	garr_betriebsmeldungen[st_config.i16_meld_startindex + 0] := FALSE;
	garr_betriebsmeldungen[st_config.i16_meld_startindex + 1] := FALSE;
	garr_betriebsmeldungen[st_config.i16_meld_startindex + 2] := FALSE;
	garr_betriebsmeldungen[st_config.i16_meld_startindex + 3] := FALSE;
	garr_betriebsmeldungen[st_config.i16_meld_startindex + 4] := FALSE;
	garr_betriebsmeldungen[st_config.i16_meld_startindex + 5] := FALSE;
	garr_betriebsmeldungen[st_config.i16_meld_startindex + 6] := FALSE;
	garr_betriebsmeldungen[st_config.i16_meld_startindex + 7] := FALSE;
	garr_betriebsmeldungen[st_config.i16_meld_startindex + 8] := FALSE;
	garr_betriebsmeldungen[st_config.i16_meld_startindex + 9] := FALSE;
	garr_betriebsmeldungen[st_config.i16_meld_startindex + 10] := FALSE;
	garr_betriebsmeldungen[st_config.i16_meld_startindex + 11] := FALSE;
	garr_betriebsmeldungen[st_config.i16_meld_startindex + 12] := FALSE;
	garr_betriebsmeldungen[st_config.i16_meld_startindex + 13] := FALSE;
	garr_betriebsmeldungen[st_config.i16_meld_startindex + 14] := FALSE;
	garr_betriebsmeldungen[st_config.i16_meld_startindex + 15] := FALSE;
	garr_betriebsmeldungen[st_config.i16_meld_startindex + 16] := FALSE;
	garr_betriebsmeldungen[st_config.i16_meld_startindex + 17] := FALSE;
	garr_betriebsmeldungen[st_config.i16_meld_startindex + 18] := FALSE;
	garr_betriebsmeldungen[st_config.i16_meld_startindex + 19] := FALSE;
END_IF
END_PROGRAM

(* POU Gemeinsamkeiten17xx/Zylinder/ST_Zylinder, ST *)
PROGRAM ST_Zylinder
VAR
	b_first_cycle 			: BOOL := TRUE;
END_VAR
IF ST_BBGen.b_lesen_komplett THEN

	ST_Datainit_Zylinder();

	(* Zylinderaufrufe *)
	zyl_wt_zentrierer_tisch.fb(
		st_config:= ,
		bw_nocken_zylinder_einfahren:= ,
		bw_nocken_zylinder_ausfahren:= ,
		uw_nocken_zylinder_einfahren:= ,
		uw_nocken_zylinder_ausfahren:= ,
		b_direkttaste_ausfahren:= ,
		b_direkttaste_mittefahren:= ,
		b_direkttaste_einfahren	:= ,
		e_druckwaechter:= ST_Betriebsfreigaben.e_druckwaechter,
		i16_betriebsart:= gi16_betriebsart,
		b_no_gesteuert_im_norm_betrieb:= ,
		st_ctrl_in:= zyl_wt_zentrierer_tisch.st_ctrl.in,
		b_masterachse_hand_dialog_aktiv:= ,
		st_visu:= visu.st_zyl,
		st_ctrl_out=> zyl_wt_zentrierer_tisch.st_ctrl.out,
		a_ventil_einfahren=> ,
		a_ventil_ausfahren=> );
	
	zyl_wt_stopper_tisch.fb(
		st_config:= ,
		bw_nocken_zylinder_einfahren:= ,
		bw_nocken_zylinder_ausfahren:= ,
		uw_nocken_zylinder_einfahren:= ,
		uw_nocken_zylinder_ausfahren:= ,
		b_direkttaste_ausfahren:= ,
		b_direkttaste_mittefahren:= ,
		b_direkttaste_einfahren	:= ,
		e_druckwaechter:= ST_Betriebsfreigaben.e_druckwaechter,
		i16_betriebsart:= gi16_betriebsart,
		b_no_gesteuert_im_norm_betrieb:= ,
		st_ctrl_in:= zyl_wt_stopper_tisch.st_ctrl.in,
		b_masterachse_hand_dialog_aktiv:= ,
		st_visu:= visu.st_zyl,
		st_ctrl_out=> zyl_wt_stopper_tisch.st_ctrl.out,
		a_ventil_einfahren=> ,
		a_ventil_ausfahren=> );
	
	zyl_wt_stopper_auslauf.fb(
		st_config:= ,
		bw_nocken_zylinder_einfahren:= ,
		bw_nocken_zylinder_ausfahren:= ,
		uw_nocken_zylinder_einfahren:= ,
		uw_nocken_zylinder_ausfahren:= ,
		b_direkttaste_ausfahren:= ,
		b_direkttaste_mittefahren:= ,
		b_direkttaste_einfahren	:= ,
		e_druckwaechter:= ST_Betriebsfreigaben.e_druckwaechter,
		i16_betriebsart:= gi16_betriebsart,
		b_no_gesteuert_im_norm_betrieb:= ,
		st_ctrl_in:= zyl_wt_stopper_auslauf.st_ctrl.in,
		b_masterachse_hand_dialog_aktiv:= ,
		st_visu:= visu.st_zyl,
		st_ctrl_out=> zyl_wt_stopper_auslauf.st_ctrl.out,
		a_ventil_einfahren=> ,
		a_ventil_ausfahren=> );
	
	zyl_hublift_rechts_lift.fb(
		st_config:= ,
		bw_nocken_zylinder_einfahren:= ,
		bw_nocken_zylinder_ausfahren:= ,
		uw_nocken_zylinder_einfahren:= ,
		uw_nocken_zylinder_ausfahren:= ,
		b_direkttaste_ausfahren:= ,
		b_direkttaste_mittefahren:= ,
		b_direkttaste_einfahren	:= ,
		e_druckwaechter:= ST_Betriebsfreigaben.e_druckwaechter,
		i16_betriebsart:= gi16_betriebsart,
		b_no_gesteuert_im_norm_betrieb:= ,
		st_ctrl_in:= zyl_hublift_rechts_lift.st_ctrl.in,
		b_masterachse_hand_dialog_aktiv:= ,
		st_visu:= visu.st_zyl,
		st_ctrl_out=> zyl_hublift_rechts_lift.st_ctrl.out,
		a_ventil_einfahren=> ,
		a_ventil_ausfahren=> );
	
	zyl_hublift_rechts_wt_einzug.fb(
		st_config:= ,
		bw_nocken_zylinder_einfahren:= ,
		bw_nocken_zylinder_ausfahren:= ,
		uw_nocken_zylinder_einfahren:= ,
		uw_nocken_zylinder_ausfahren:= ,
		b_direkttaste_ausfahren:= ,
		b_direkttaste_mittefahren:= ,
		b_direkttaste_einfahren	:= ,
		e_druckwaechter:= ST_Betriebsfreigaben.e_druckwaechter,
		i16_betriebsart:= gi16_betriebsart,
		b_no_gesteuert_im_norm_betrieb:= ,
		st_ctrl_in:= zyl_hublift_rechts_wt_einzug.st_ctrl.in,
		b_masterachse_hand_dialog_aktiv:= ,
		st_visu:= visu.st_zyl,
		st_ctrl_out=> zyl_hublift_rechts_wt_einzug.st_ctrl.out,
		a_ventil_einfahren=> ,
		a_ventil_ausfahren=> );
	
	zyl_hublift_rechts_wt_klinke.fb(
		st_config:= ,
		bw_nocken_zylinder_einfahren:= ,
		bw_nocken_zylinder_ausfahren:= ,
		uw_nocken_zylinder_einfahren:= ,
		uw_nocken_zylinder_ausfahren:= ,
		b_direkttaste_ausfahren:= ,
		b_direkttaste_mittefahren:= ,
		b_direkttaste_einfahren	:= ,
		e_druckwaechter:= ST_Betriebsfreigaben.e_druckwaechter,
		i16_betriebsart:= gi16_betriebsart,
		b_no_gesteuert_im_norm_betrieb:= ,
		st_ctrl_in:= zyl_hublift_rechts_wt_klinke.st_ctrl.in,
		b_masterachse_hand_dialog_aktiv:= ,
		st_visu:= visu.st_zyl,
		st_ctrl_out=> zyl_hublift_rechts_wt_klinke.st_ctrl.out,
		a_ventil_einfahren=> ,
		a_ventil_ausfahren=> );
	
	zyl_hublift_links_lift.fb(
		st_config:= ,
		bw_nocken_zylinder_einfahren:= ,
		bw_nocken_zylinder_ausfahren:= ,
		uw_nocken_zylinder_einfahren:= ,
		uw_nocken_zylinder_ausfahren:= ,
		b_direkttaste_ausfahren:= ,
		b_direkttaste_mittefahren:= ,
		b_direkttaste_einfahren	:= ,
		e_druckwaechter:= ST_Betriebsfreigaben.e_druckwaechter,
		i16_betriebsart:= gi16_betriebsart,
		b_no_gesteuert_im_norm_betrieb:= ,
		st_ctrl_in:= zyl_hublift_links_lift.st_ctrl.in,
		b_masterachse_hand_dialog_aktiv:= ,
		st_visu:= visu.st_zyl,
		st_ctrl_out=> zyl_hublift_links_lift.st_ctrl.out,
		a_ventil_einfahren=> ,
		a_ventil_ausfahren=> );
	
	zyl_hublift_links_wt_einzug.fb(
		st_config:= ,
		bw_nocken_zylinder_einfahren:= ,
		bw_nocken_zylinder_ausfahren:= ,
		uw_nocken_zylinder_einfahren:= ,
		uw_nocken_zylinder_ausfahren:= ,
		b_direkttaste_ausfahren:= ,
		b_direkttaste_mittefahren:= ,
		b_direkttaste_einfahren	:= ,
		e_druckwaechter:= ST_Betriebsfreigaben.e_druckwaechter,
		i16_betriebsart:= gi16_betriebsart,
		b_no_gesteuert_im_norm_betrieb:= ,
		st_ctrl_in:= zyl_hublift_links_wt_einzug.st_ctrl.in,
		b_masterachse_hand_dialog_aktiv:= ,
		st_visu:= visu.st_zyl,
		st_ctrl_out=> zyl_hublift_links_wt_einzug.st_ctrl.out,
		a_ventil_einfahren=> ,
		a_ventil_ausfahren=> );
	
	zyl_hublift_links_wt_klinke.fb(
		st_config:= ,
		bw_nocken_zylinder_einfahren:= ,
		bw_nocken_zylinder_ausfahren:= ,
		uw_nocken_zylinder_einfahren:= ,
		uw_nocken_zylinder_ausfahren:= ,
		b_direkttaste_ausfahren:= ,
		b_direkttaste_mittefahren:= ,
		b_direkttaste_einfahren	:= ,
		e_druckwaechter:= ST_Betriebsfreigaben.e_druckwaechter,
		i16_betriebsart:= gi16_betriebsart,
		b_no_gesteuert_im_norm_betrieb:= ,
		st_ctrl_in:= zyl_hublift_links_wt_klinke.st_ctrl.in,
		b_masterachse_hand_dialog_aktiv:= ,
		st_visu:= visu.st_zyl,
		st_ctrl_out=> zyl_hublift_links_wt_klinke.st_ctrl.out,
		a_ventil_einfahren=> ,
		a_ventil_ausfahren=> );
	
	zyl_hublift_links_stopper.fb(
		st_config:= ,
		bw_nocken_zylinder_einfahren:= ,
		bw_nocken_zylinder_ausfahren:= ,
		uw_nocken_zylinder_einfahren:= ,
		uw_nocken_zylinder_ausfahren:= ,
		b_direkttaste_ausfahren:= ,
		b_direkttaste_mittefahren:= ,
		b_direkttaste_einfahren	:= ,
		e_druckwaechter:= ST_Betriebsfreigaben.e_druckwaechter,
		i16_betriebsart:= gi16_betriebsart,
		b_no_gesteuert_im_norm_betrieb:= ,
		st_ctrl_in:= zyl_hublift_links_stopper.st_ctrl.in,
		b_masterachse_hand_dialog_aktiv:= ,
		st_visu:= visu.st_zyl,
		st_ctrl_out=> zyl_hublift_links_stopper.st_ctrl.out,
		a_ventil_einfahren=> ,
		a_ventil_ausfahren=> );
	
	zyl_hublift_links_eingriffschutz.fb(
		st_config:= ,
		bw_nocken_zylinder_einfahren:= ,
		bw_nocken_zylinder_ausfahren:= ,
		uw_nocken_zylinder_einfahren:= ,
		uw_nocken_zylinder_ausfahren:= ,
		b_direkttaste_ausfahren:= ,
		b_direkttaste_mittefahren:= ,
		b_direkttaste_einfahren	:= ,
		e_druckwaechter:= ST_Betriebsfreigaben.e_druckwaechter,
		i16_betriebsart:= gi16_betriebsart,
		b_no_gesteuert_im_norm_betrieb:= ,
		st_ctrl_in:= zyl_hublift_links_eingriffschutz.st_ctrl.in,
		b_masterachse_hand_dialog_aktiv:= ,
		st_visu:= visu.st_zyl,
		st_ctrl_out=> zyl_hublift_links_eingriffschutz.st_ctrl.out,
		a_ventil_einfahren=> ,
		a_ventil_ausfahren=> );
	
	CASE gst_datensatz.st_md.i16_typ_zelle OF
		KEINE_ZELLE:
			;
	
		BESTUECKZELLE_1700:
			zyl_bawe_faenger_li.fb.st_config.b_aktiv := NOT gst_datensatz.st_md.b_wt_transport_simulation;
			zyl_bawe_faenger_li.fb(
				st_config:= ,
				bw_nocken_zylinder_einfahren:= ,
				bw_nocken_zylinder_ausfahren:= ,
				uw_nocken_zylinder_einfahren:= ,
				uw_nocken_zylinder_ausfahren:= ,
				b_direkttaste_ausfahren:= ,
				b_direkttaste_mittefahren:= ,
				b_direkttaste_einfahren	:= ,
				e_druckwaechter:= ST_Betriebsfreigaben.e_druckwaechter,
				i16_betriebsart:= gi16_betriebsart,
				b_no_gesteuert_im_norm_betrieb:= ,
				st_ctrl_in:= zyl_bawe_faenger_li.st_ctrl.in,
				b_masterachse_hand_dialog_aktiv:= ,
				st_visu:= visu.st_zyl,
				st_ctrl_out=> zyl_bawe_faenger_li.st_ctrl.out,
				a_ventil_einfahren=> ,
				a_ventil_ausfahren=> );
	
			zyl_bawe_faenger_re.fb.st_config.b_aktiv := NOT gst_datensatz.st_md.b_wt_transport_simulation;
			zyl_bawe_faenger_re.fb(
				st_config:= ,
				bw_nocken_zylinder_einfahren:= ,
				bw_nocken_zylinder_ausfahren:= ,
				uw_nocken_zylinder_einfahren:= ,
				uw_nocken_zylinder_ausfahren:= ,
				b_direkttaste_ausfahren:= ,
				b_direkttaste_mittefahren:= ,
				b_direkttaste_einfahren	:= ,
				e_druckwaechter:= ST_Betriebsfreigaben.e_druckwaechter,
				i16_betriebsart:= gi16_betriebsart,
				b_no_gesteuert_im_norm_betrieb:= ,
				st_ctrl_in:= zyl_bawe_faenger_re.st_ctrl.in,
				b_masterachse_hand_dialog_aktiv:= ,
				st_visu:= visu.st_zyl,
				st_ctrl_out=> zyl_bawe_faenger_re.st_ctrl.out,
				a_ventil_einfahren=> ,
				a_ventil_ausfahren=> );
	
			zyl_bawe_halter_li.fb.st_config.b_aktiv := NOT gst_datensatz.st_md.b_wt_transport_simulation;
			zyl_bawe_halter_li.fb(
				st_config:= ,
				bw_nocken_zylinder_einfahren:= ,
				bw_nocken_zylinder_ausfahren:= ,
				uw_nocken_zylinder_einfahren:= ,
				uw_nocken_zylinder_ausfahren:= ,
				b_direkttaste_ausfahren:= ,
				b_direkttaste_mittefahren:= ,
				b_direkttaste_einfahren	:= ,
				e_druckwaechter:= ST_Betriebsfreigaben.e_druckwaechter,
				i16_betriebsart:= gi16_betriebsart,
				b_no_gesteuert_im_norm_betrieb:= ,
				st_ctrl_in:= zyl_bawe_halter_li.st_ctrl.in,
				b_masterachse_hand_dialog_aktiv:= ,
				st_visu:= visu.st_zyl,
				st_ctrl_out=> zyl_bawe_halter_li.st_ctrl.out,
				a_ventil_einfahren=> ,
				a_ventil_ausfahren=> );
	
			zyl_bawe_halter_re.fb.st_config.b_aktiv := NOT gst_datensatz.st_md.b_wt_transport_simulation;
			zyl_bawe_halter_re.fb(
				st_config:= ,
				bw_nocken_zylinder_einfahren:= ,
				bw_nocken_zylinder_ausfahren:= ,
				uw_nocken_zylinder_einfahren:= ,
				uw_nocken_zylinder_ausfahren:= ,
				b_direkttaste_ausfahren:= ,
				b_direkttaste_mittefahren:= ,
				b_direkttaste_einfahren	:= ,
				e_druckwaechter:= ST_Betriebsfreigaben.e_druckwaechter,
				i16_betriebsart:= gi16_betriebsart,
				b_no_gesteuert_im_norm_betrieb:= ,
				st_ctrl_in:= zyl_bawe_halter_re.st_ctrl.in,
				b_masterachse_hand_dialog_aktiv:= ,
				st_visu:= visu.st_zyl,
				st_ctrl_out=> zyl_bawe_halter_re.st_ctrl.out,
				a_ventil_einfahren=> ,
				a_ventil_ausfahren=> );
	
			zyl_bawe_querschub.fb.st_config.b_aktiv := NOT gst_datensatz.st_md.b_wt_transport_simulation;
			zyl_bawe_querschub.fb(
				st_config:= ,
				bw_nocken_zylinder_einfahren:= ,
				bw_nocken_zylinder_ausfahren:= ,
				uw_nocken_zylinder_einfahren:= ,
				uw_nocken_zylinder_ausfahren:= ,
				b_direkttaste_ausfahren:= ,
				b_direkttaste_mittefahren:= ,
				b_direkttaste_einfahren	:= ,
				e_druckwaechter:= ST_Betriebsfreigaben.e_druckwaechter,
				i16_betriebsart:= gi16_betriebsart,
				b_no_gesteuert_im_norm_betrieb:= ,
				st_ctrl_in:= zyl_bawe_querschub.st_ctrl.in,
				b_masterachse_hand_dialog_aktiv:= ,
				st_visu:= visu.st_zyl,
				st_ctrl_out=> zyl_bawe_querschub.st_ctrl.out,
				a_ventil_einfahren=> ,
				a_ventil_ausfahren=> );
	
			zyl_bawe_vorschub.fb.st_config.b_aktiv := NOT gst_datensatz.st_md.b_wt_transport_simulation;
			zyl_bawe_vorschub.fb(
				st_config:= ,
				bw_nocken_zylinder_einfahren:= ,
				bw_nocken_zylinder_ausfahren:= ,
				uw_nocken_zylinder_einfahren:= ,
				uw_nocken_zylinder_ausfahren:= ,
				b_direkttaste_ausfahren:= ,
				b_direkttaste_mittefahren:= ,
				b_direkttaste_einfahren	:= ,
				e_druckwaechter:= ST_Betriebsfreigaben.e_druckwaechter,
				i16_betriebsart:= gi16_betriebsart,
				b_no_gesteuert_im_norm_betrieb:= ,
				st_ctrl_in:= zyl_bawe_vorschub.st_ctrl.in,
				b_masterachse_hand_dialog_aktiv:= ,
				st_visu:= visu.st_zyl,
				st_ctrl_out=> zyl_bawe_vorschub.st_ctrl.out,
				a_ventil_einfahren=> a_zyl_vorschub_einfahren,
				a_ventil_ausfahren=> a_zyl_vorschub_ausfahren);
			
			zyl_haspel_li_heben.fb(
				st_config:= ,
				bw_nocken_zylinder_einfahren:= ,
				bw_nocken_zylinder_ausfahren:= ,
				uw_nocken_zylinder_einfahren:= ,
				uw_nocken_zylinder_ausfahren:= ,
				b_direkttaste_ausfahren:= ,
				b_direkttaste_mittefahren:= ,
				b_direkttaste_einfahren	:= ,
				e_druckwaechter:= ST_Betriebsfreigaben.e_druckwaechter,
				i16_betriebsart:= gi16_betriebsart,
				b_no_gesteuert_im_norm_betrieb:= ,
				st_ctrl_in:= zyl_haspel_li_heben.st_ctrl.in,
				b_masterachse_hand_dialog_aktiv:= ,
				st_visu:= visu.st_zyl,
				st_ctrl_out=> zyl_haspel_li_heben.st_ctrl.out,
				a_ventil_einfahren=> ,
				a_ventil_ausfahren=> );
	
			zyl_haspel_li_abspulen.fb(
				st_config:= ,
				bw_nocken_zylinder_einfahren:= ,
				bw_nocken_zylinder_ausfahren:= ,
				uw_nocken_zylinder_einfahren:= ,
				uw_nocken_zylinder_ausfahren:= ,
				b_direkttaste_ausfahren:= ,
				b_direkttaste_mittefahren:= ,
				b_direkttaste_einfahren	:= ,
				e_druckwaechter:= ST_Betriebsfreigaben.e_druckwaechter,
				i16_betriebsart:= gi16_betriebsart,
				b_no_gesteuert_im_norm_betrieb:= ,
				st_ctrl_in:= zyl_haspel_li_abspulen.st_ctrl.in,
				b_masterachse_hand_dialog_aktiv:= ,
				st_visu:= visu.st_zyl,
				st_ctrl_out=> zyl_haspel_li_abspulen.st_ctrl.out,
				a_ventil_einfahren=> ,
				a_ventil_ausfahren=> );
			
			zyl_haspel_li_sperren.fb(
				st_config:= ,
				bw_nocken_zylinder_einfahren:= ,
				bw_nocken_zylinder_ausfahren:= ,
				uw_nocken_zylinder_einfahren:= ,
				uw_nocken_zylinder_ausfahren:= ,
				b_direkttaste_ausfahren:= ,
				b_direkttaste_mittefahren:= ,
				b_direkttaste_einfahren	:= ,
				e_druckwaechter:= ST_Betriebsfreigaben.e_druckwaechter,
				i16_betriebsart:= gi16_betriebsart,
				b_no_gesteuert_im_norm_betrieb:= ,
				st_ctrl_in:= zyl_haspel_li_sperren.st_ctrl.in,
				b_masterachse_hand_dialog_aktiv:= ,
				st_visu:= visu.st_zyl,
				st_ctrl_out=> zyl_haspel_li_sperren.st_ctrl.out,
				a_ventil_einfahren=> ,
				a_ventil_ausfahren=> );
			
			zyl_haspel_re_heben.fb(
				st_config:= ,
				bw_nocken_zylinder_einfahren:= ,
				bw_nocken_zylinder_ausfahren:= ,
				uw_nocken_zylinder_einfahren:= ,
				uw_nocken_zylinder_ausfahren:= ,
				b_direkttaste_ausfahren:= ,
				b_direkttaste_mittefahren:= ,
				b_direkttaste_einfahren	:= ,
				e_druckwaechter:= ST_Betriebsfreigaben.e_druckwaechter,
				i16_betriebsart:= gi16_betriebsart,
				b_no_gesteuert_im_norm_betrieb:= ,
				st_ctrl_in:= zyl_haspel_re_heben.st_ctrl.in,
				b_masterachse_hand_dialog_aktiv:= ,
				st_visu:= visu.st_zyl,
				st_ctrl_out=> zyl_haspel_re_heben.st_ctrl.out,
				a_ventil_einfahren=> ,
				a_ventil_ausfahren=> );
			
			zyl_haspel_re_abspulen.fb(
				st_config:= ,
				bw_nocken_zylinder_einfahren:= ,
				bw_nocken_zylinder_ausfahren:= ,
				uw_nocken_zylinder_einfahren:= ,
				uw_nocken_zylinder_ausfahren:= ,
				b_direkttaste_ausfahren:= ,
				b_direkttaste_mittefahren:= ,
				b_direkttaste_einfahren	:= ,
				e_druckwaechter:= ST_Betriebsfreigaben.e_druckwaechter,
				i16_betriebsart:= gi16_betriebsart,
				b_no_gesteuert_im_norm_betrieb:= ,
				st_ctrl_in:= zyl_haspel_re_abspulen.st_ctrl.in,
				b_masterachse_hand_dialog_aktiv:= ,
				st_visu:= visu.st_zyl,
				st_ctrl_out=> zyl_haspel_re_abspulen.st_ctrl.out,
				a_ventil_einfahren=> ,
				a_ventil_ausfahren=> );
			
			zyl_haspel_re_sperren.fb(
				st_config:= ,
				bw_nocken_zylinder_einfahren:= ,
				bw_nocken_zylinder_ausfahren:= ,
				uw_nocken_zylinder_einfahren:= ,
				uw_nocken_zylinder_ausfahren:= ,
				b_direkttaste_ausfahren:= ,
				b_direkttaste_mittefahren:= ,
				b_direkttaste_einfahren	:= ,
				e_druckwaechter:= ST_Betriebsfreigaben.e_druckwaechter,
				i16_betriebsart:= gi16_betriebsart,
				b_no_gesteuert_im_norm_betrieb:= ,
				st_ctrl_in:= zyl_haspel_re_sperren.st_ctrl.in,
				b_masterachse_hand_dialog_aktiv:= ,
				st_visu:= visu.st_zyl,
				st_ctrl_out=> zyl_haspel_re_sperren.st_ctrl.out,
				a_ventil_einfahren=> ,
				a_ventil_ausfahren=> );
			
			zyl_haspel_verschieben.fb(
				st_config:= ,
				bw_nocken_zylinder_einfahren:= ,
				bw_nocken_zylinder_ausfahren:= ,
				uw_nocken_zylinder_einfahren:= ,
				uw_nocken_zylinder_ausfahren:= ,
				b_direkttaste_ausfahren:= ,
				b_direkttaste_mittefahren:= ,
				b_direkttaste_einfahren	:= ,
				e_druckwaechter:= ST_Betriebsfreigaben.e_druckwaechter,
				i16_betriebsart:= gi16_betriebsart,
				b_no_gesteuert_im_norm_betrieb:= ,
				st_ctrl_in:= zyl_haspel_verschieben.st_ctrl.in,
				b_masterachse_hand_dialog_aktiv:= ,
				st_visu:= visu.st_zyl,
				st_ctrl_out=> zyl_haspel_verschieben.st_ctrl.out,
				a_ventil_einfahren=> ,
				a_ventil_ausfahren=> );

			zyl_bandeinzuege_verschieben.fb(
				st_config:= ,
				bw_nocken_zylinder_einfahren:= ,
				bw_nocken_zylinder_ausfahren:= ,
				uw_nocken_zylinder_einfahren:= ,
				uw_nocken_zylinder_ausfahren:= ,
				b_direkttaste_ausfahren:= ,
				b_direkttaste_mittefahren:= ,
				b_direkttaste_einfahren	:= ,
				e_druckwaechter:= ST_Betriebsfreigaben.e_druckwaechter,
				i16_betriebsart:= gi16_betriebsart,
				b_no_gesteuert_im_norm_betrieb:= ,
				st_ctrl_in:= zyl_bandeinzuege_verschieben.st_ctrl.in,
				b_masterachse_hand_dialog_aktiv:= ,
				st_visu:= visu.st_zyl,
				st_ctrl_out=> zyl_bandeinzuege_verschieben.st_ctrl.out,
				a_ventil_einfahren=> ,
				a_ventil_ausfahren=> );
	

		(*	zyl_Indexier_Bestueckpos.fb.st_config.b_aktiv := NOT gst_datensatz.st_md.b_wt_transport_simulation;*)
			zyl_Indexier_Bestueckpos.fb(
				st_config:= ,
				bw_nocken_zylinder_einfahren:= ,
				bw_nocken_zylinder_ausfahren:= ,
				uw_nocken_zylinder_einfahren:= ,
				uw_nocken_zylinder_ausfahren:= ,
				b_direkttaste_ausfahren:= ,
				b_direkttaste_mittefahren:= ,
				b_direkttaste_einfahren	:= ,
				e_druckwaechter:= ST_Betriebsfreigaben.e_druckwaechter,
				i16_betriebsart:= gi16_betriebsart,
				b_no_gesteuert_im_norm_betrieb:= ,
				st_ctrl_in:= zyl_Indexier_Bestueckpos.st_ctrl.in,
				b_masterachse_hand_dialog_aktiv:= ,
				st_visu:= visu.st_zyl,
				st_ctrl_out=> zyl_Indexier_Bestueckpos.st_ctrl.out,
				a_ventil_einfahren=> ,
				a_ventil_ausfahren=> );
	
		(*	zyl_Indexier_Einlauf.fb.st_config.b_aktiv := NOT gst_datensatz.st_md.b_wt_transport_simulation;*)
			zyl_Indexier_Einlauf.fb(
				st_config:= ,
				bw_nocken_zylinder_einfahren:= ,
				bw_nocken_zylinder_ausfahren:= ,
				uw_nocken_zylinder_einfahren:= ,
				uw_nocken_zylinder_ausfahren:= ,
				b_direkttaste_ausfahren:= ,
				b_direkttaste_mittefahren:= ,
				b_direkttaste_einfahren	:= ,
				e_druckwaechter:= ST_Betriebsfreigaben.e_druckwaechter,
				i16_betriebsart:= gi16_betriebsart,
				b_no_gesteuert_im_norm_betrieb:= ,
				st_ctrl_in:= zyl_Indexier_Einlauf.st_ctrl.in,
				b_masterachse_hand_dialog_aktiv:= ,
				st_visu:= visu.st_zyl,
				st_ctrl_out=> zyl_Indexier_Einlauf.st_ctrl.out,
				a_ventil_einfahren=> ,
				a_ventil_ausfahren=> );

		BESTUECKZELLE_1720:
			zyl_wt_stopper_einlauf.fb(
				st_config:= ,
				bw_nocken_zylinder_einfahren:= ,
				bw_nocken_zylinder_ausfahren:= ,
				uw_nocken_zylinder_einfahren:= ,
				uw_nocken_zylinder_ausfahren:= ,
				b_direkttaste_ausfahren:= ,
				b_direkttaste_mittefahren:= ,
				b_direkttaste_einfahren	:= ,
				e_druckwaechter:= ST_Betriebsfreigaben.e_druckwaechter,
				i16_betriebsart:= gi16_betriebsart,
				b_no_gesteuert_im_norm_betrieb:= ,
				st_ctrl_in:= zyl_wt_stopper_einlauf.st_ctrl.in,
				b_masterachse_hand_dialog_aktiv:= ,
				st_visu:= visu.st_zyl,
				st_ctrl_out=> zyl_wt_stopper_einlauf.st_ctrl.out,
				a_ventil_einfahren=> ,
				a_ventil_ausfahren=> );
	
			zyl_haspel_li_heben.fb(
				st_config:= ,
				bw_nocken_zylinder_einfahren:= ,
				bw_nocken_zylinder_ausfahren:= ,
				uw_nocken_zylinder_einfahren:= ,
				uw_nocken_zylinder_ausfahren:= ,
				b_direkttaste_ausfahren:= ,
				b_direkttaste_mittefahren:= ,
				b_direkttaste_einfahren	:= ,
				e_druckwaechter:= ST_Betriebsfreigaben.e_druckwaechter,
				i16_betriebsart:= gi16_betriebsart,
				b_no_gesteuert_im_norm_betrieb:= ,
				st_ctrl_in:= zyl_haspel_li_heben.st_ctrl.in,
				b_masterachse_hand_dialog_aktiv:= ,
				st_visu:= visu.st_zyl,
				st_ctrl_out=> zyl_haspel_li_heben.st_ctrl.out,
				a_ventil_einfahren=> ,
				a_ventil_ausfahren=> );
			
			zyl_haspel_li_abspulen.fb(
				st_config:= ,
				bw_nocken_zylinder_einfahren:= ,
				bw_nocken_zylinder_ausfahren:= ,
				uw_nocken_zylinder_einfahren:= ,
				uw_nocken_zylinder_ausfahren:= ,
				b_direkttaste_ausfahren:= ,
				b_direkttaste_mittefahren:= ,
				b_direkttaste_einfahren	:= ,
				e_druckwaechter:= ST_Betriebsfreigaben.e_druckwaechter,
				i16_betriebsart:= gi16_betriebsart,
				b_no_gesteuert_im_norm_betrieb:= ,
				st_ctrl_in:= zyl_haspel_li_abspulen.st_ctrl.in,
				b_masterachse_hand_dialog_aktiv:= ,
				st_visu:= visu.st_zyl,
				st_ctrl_out=> zyl_haspel_li_abspulen.st_ctrl.out,
				a_ventil_einfahren=> ,
				a_ventil_ausfahren=> );
			
			zyl_haspel_li_sperren.fb(
				st_config:= ,
				bw_nocken_zylinder_einfahren:= ,
				bw_nocken_zylinder_ausfahren:= ,
				uw_nocken_zylinder_einfahren:= ,
				uw_nocken_zylinder_ausfahren:= ,
				b_direkttaste_ausfahren:= ,
				b_direkttaste_mittefahren:= ,
				b_direkttaste_einfahren	:= ,
				e_druckwaechter:= ST_Betriebsfreigaben.e_druckwaechter,
				i16_betriebsart:= gi16_betriebsart,
				b_no_gesteuert_im_norm_betrieb:= ,
				st_ctrl_in:= zyl_haspel_li_sperren.st_ctrl.in,
				b_masterachse_hand_dialog_aktiv:= ,
				st_visu:= visu.st_zyl,
				st_ctrl_out=> zyl_haspel_li_sperren.st_ctrl.out,
				a_ventil_einfahren=> ,
				a_ventil_ausfahren=> );
			
			zyl_haspel_re_heben.fb(
				st_config:= ,
				bw_nocken_zylinder_einfahren:= ,
				bw_nocken_zylinder_ausfahren:= ,
				uw_nocken_zylinder_einfahren:= ,
				uw_nocken_zylinder_ausfahren:= ,
				b_direkttaste_ausfahren:= ,
				b_direkttaste_mittefahren:= ,
				b_direkttaste_einfahren	:= ,
				e_druckwaechter:= ST_Betriebsfreigaben.e_druckwaechter,
				i16_betriebsart:= gi16_betriebsart,
				b_no_gesteuert_im_norm_betrieb:= ,
				st_ctrl_in:= zyl_haspel_re_heben.st_ctrl.in,
				b_masterachse_hand_dialog_aktiv:= ,
				st_visu:= visu.st_zyl,
				st_ctrl_out=> zyl_haspel_re_heben.st_ctrl.out,
				a_ventil_einfahren=> ,
				a_ventil_ausfahren=> );
			
			zyl_haspel_re_abspulen.fb(
				st_config:= ,
				bw_nocken_zylinder_einfahren:= ,
				bw_nocken_zylinder_ausfahren:= ,
				uw_nocken_zylinder_einfahren:= ,
				uw_nocken_zylinder_ausfahren:= ,
				b_direkttaste_ausfahren:= ,
				b_direkttaste_mittefahren:= ,
				b_direkttaste_einfahren	:= ,
				e_druckwaechter:= ST_Betriebsfreigaben.e_druckwaechter,
				i16_betriebsart:= gi16_betriebsart,
				b_no_gesteuert_im_norm_betrieb:= ,
				st_ctrl_in:= zyl_haspel_re_abspulen.st_ctrl.in,
				b_masterachse_hand_dialog_aktiv:= ,
				st_visu:= visu.st_zyl,
				st_ctrl_out=> zyl_haspel_re_abspulen.st_ctrl.out,
				a_ventil_einfahren=> ,
				a_ventil_ausfahren=> );
			
			zyl_haspel_re_sperren.fb(
				st_config:= ,
				bw_nocken_zylinder_einfahren:= ,
				bw_nocken_zylinder_ausfahren:= ,
				uw_nocken_zylinder_einfahren:= ,
				uw_nocken_zylinder_ausfahren:= ,
				b_direkttaste_ausfahren:= ,
				b_direkttaste_mittefahren:= ,
				b_direkttaste_einfahren	:= ,
				e_druckwaechter:= ST_Betriebsfreigaben.e_druckwaechter,
				i16_betriebsart:= gi16_betriebsart,
				b_no_gesteuert_im_norm_betrieb:= ,
				st_ctrl_in:= zyl_haspel_re_sperren.st_ctrl.in,
				b_masterachse_hand_dialog_aktiv:= ,
				st_visu:= visu.st_zyl,
				st_ctrl_out=> zyl_haspel_re_sperren.st_ctrl.out,
				a_ventil_einfahren=> ,
				a_ventil_ausfahren=> );
	
			zyl_bawe_halter_li.fb.st_config.b_aktiv := NOT gst_datensatz.st_md.b_wt_transport_simulation;
			zyl_bawe_halter_li.fb(
				st_config:= ,
				bw_nocken_zylinder_einfahren:= ,
				bw_nocken_zylinder_ausfahren:= ,
				uw_nocken_zylinder_einfahren:= ,
				uw_nocken_zylinder_ausfahren:= ,
				b_direkttaste_ausfahren:= ,
				b_direkttaste_mittefahren:= ,
				b_direkttaste_einfahren	:= ,
				e_druckwaechter:= ST_Betriebsfreigaben.e_druckwaechter,
				i16_betriebsart:= gi16_betriebsart,
				b_no_gesteuert_im_norm_betrieb:= ,
				st_ctrl_in:= zyl_bawe_halter_li.st_ctrl.in,
				b_masterachse_hand_dialog_aktiv:= ,
				st_visu:= visu.st_zyl,
				st_ctrl_out=> zyl_bawe_halter_li.st_ctrl.out,
				a_ventil_einfahren=> ,
				a_ventil_ausfahren=> );
	
			zyl_bawe_halter_re.fb.st_config.b_aktiv := NOT gst_datensatz.st_md.b_wt_transport_simulation;
			zyl_bawe_halter_re.fb(
				st_config:= ,
				bw_nocken_zylinder_einfahren:= ,
				bw_nocken_zylinder_ausfahren:= ,
				uw_nocken_zylinder_einfahren:= ,
				uw_nocken_zylinder_ausfahren:= ,
				b_direkttaste_ausfahren:= ,
				b_direkttaste_mittefahren:= ,
				b_direkttaste_einfahren	:= ,
				e_druckwaechter:= ST_Betriebsfreigaben.e_druckwaechter,
				i16_betriebsart:= gi16_betriebsart,
				b_no_gesteuert_im_norm_betrieb:= ,
				st_ctrl_in:= zyl_bawe_halter_re.st_ctrl.in,
				b_masterachse_hand_dialog_aktiv:= ,
				st_visu:= visu.st_zyl,
				st_ctrl_out=> zyl_bawe_halter_re.st_ctrl.out,
				a_ventil_einfahren=> ,
				a_ventil_ausfahren=> );
	
		RASTERFOLIE:
			zyl_haspel_li_heben.fb(
				st_config:= ,
				bw_nocken_zylinder_einfahren:= ,
				bw_nocken_zylinder_ausfahren:= ,
				uw_nocken_zylinder_einfahren:= ,
				uw_nocken_zylinder_ausfahren:= ,
				b_direkttaste_ausfahren:= ,
				b_direkttaste_mittefahren:= ,
				b_direkttaste_einfahren	:= ,
				e_druckwaechter:= ST_Betriebsfreigaben.e_druckwaechter,
				i16_betriebsart:= gi16_betriebsart,
				b_no_gesteuert_im_norm_betrieb:= ,
				st_ctrl_in:= zyl_haspel_li_heben.st_ctrl.in,
				b_masterachse_hand_dialog_aktiv:= ,
				st_visu:= visu.st_zyl,
				st_ctrl_out=> zyl_haspel_li_heben.st_ctrl.out,
				a_ventil_einfahren=> ,
				a_ventil_ausfahren=> );
			
			zyl_haspel_li_abspulen.fb(
				st_config:= ,
				bw_nocken_zylinder_einfahren:= ,
				bw_nocken_zylinder_ausfahren:= ,
				uw_nocken_zylinder_einfahren:= ,
				uw_nocken_zylinder_ausfahren:= ,
				b_direkttaste_ausfahren:= ,
				b_direkttaste_mittefahren:= ,
				b_direkttaste_einfahren	:= ,
				e_druckwaechter:= ST_Betriebsfreigaben.e_druckwaechter,
				i16_betriebsart:= gi16_betriebsart,
				b_no_gesteuert_im_norm_betrieb:= ,
				st_ctrl_in:= zyl_haspel_li_abspulen.st_ctrl.in,
				b_masterachse_hand_dialog_aktiv:= ,
				st_visu:= visu.st_zyl,
				st_ctrl_out=> zyl_haspel_li_abspulen.st_ctrl.out,
				a_ventil_einfahren=> ,
				a_ventil_ausfahren=> );
	
			zyl_haspel_li_sperren.fb(
				st_config:= ,
				bw_nocken_zylinder_einfahren:= ,
				bw_nocken_zylinder_ausfahren:= ,
				uw_nocken_zylinder_einfahren:= ,
				uw_nocken_zylinder_ausfahren:= ,
				b_direkttaste_ausfahren:= ,
				b_direkttaste_mittefahren:= ,
				b_direkttaste_einfahren	:= ,
				e_druckwaechter:= ST_Betriebsfreigaben.e_druckwaechter,
				i16_betriebsart:= gi16_betriebsart,
				b_no_gesteuert_im_norm_betrieb:= ,
				st_ctrl_in:= zyl_haspel_li_sperren.st_ctrl.in,
				b_masterachse_hand_dialog_aktiv:= ,
				st_visu:= visu.st_zyl,
				st_ctrl_out=> zyl_haspel_li_sperren.st_ctrl.out,
				a_ventil_einfahren=> ,
				a_ventil_ausfahren=> );
			
			zyl_haspel_re_heben.fb(
				st_config:= ,
				bw_nocken_zylinder_einfahren:= ,
				bw_nocken_zylinder_ausfahren:= ,
				uw_nocken_zylinder_einfahren:= ,
				uw_nocken_zylinder_ausfahren:= ,
				b_direkttaste_ausfahren:= ,
				b_direkttaste_mittefahren:= ,
				b_direkttaste_einfahren	:= ,
				e_druckwaechter:= ST_Betriebsfreigaben.e_druckwaechter,
				i16_betriebsart:= gi16_betriebsart,
				b_no_gesteuert_im_norm_betrieb:= ,
				st_ctrl_in:= zyl_haspel_re_heben.st_ctrl.in,
				b_masterachse_hand_dialog_aktiv:= ,
				st_visu:= visu.st_zyl,
				st_ctrl_out=> zyl_haspel_re_heben.st_ctrl.out,
				a_ventil_einfahren=> ,
				a_ventil_ausfahren=> );
			
			zyl_haspel_re_abspulen.fb(
				st_config:= ,
				bw_nocken_zylinder_einfahren:= ,
				bw_nocken_zylinder_ausfahren:= ,
				uw_nocken_zylinder_einfahren:= ,
				uw_nocken_zylinder_ausfahren:= ,
				b_direkttaste_ausfahren:= ,
				b_direkttaste_mittefahren:= ,
				b_direkttaste_einfahren	:= ,
				e_druckwaechter:= ST_Betriebsfreigaben.e_druckwaechter,
				i16_betriebsart:= gi16_betriebsart,
				b_no_gesteuert_im_norm_betrieb:= ,
				st_ctrl_in:= zyl_haspel_re_abspulen.st_ctrl.in,
				b_masterachse_hand_dialog_aktiv:= ,
				st_visu:= visu.st_zyl,
				st_ctrl_out=> zyl_haspel_re_abspulen.st_ctrl.out,
				a_ventil_einfahren=> ,
				a_ventil_ausfahren=> );
			
			zyl_haspel_re_sperren.fb(
				st_config:= ,
				bw_nocken_zylinder_einfahren:= ,
				bw_nocken_zylinder_ausfahren:= ,
				uw_nocken_zylinder_einfahren:= ,
				uw_nocken_zylinder_ausfahren:= ,
				b_direkttaste_ausfahren:= ,
				b_direkttaste_mittefahren:= ,
				b_direkttaste_einfahren	:= ,
				e_druckwaechter:= ST_Betriebsfreigaben.e_druckwaechter,
				i16_betriebsart:= gi16_betriebsart,
				b_no_gesteuert_im_norm_betrieb:= ,
				st_ctrl_in:= zyl_haspel_re_sperren.st_ctrl.in,
				b_masterachse_hand_dialog_aktiv:= ,
				st_visu:= visu.st_zyl,
				st_ctrl_out=> zyl_haspel_re_sperren.st_ctrl.out,
				a_ventil_einfahren=> ,
				a_ventil_ausfahren=> );
			
			zyl_haspel_verschieben.fb(
				st_config:= ,
				bw_nocken_zylinder_einfahren:= ,
				bw_nocken_zylinder_ausfahren:= ,
				uw_nocken_zylinder_einfahren:= ,
				uw_nocken_zylinder_ausfahren:= ,
				b_direkttaste_ausfahren:= ,
				b_direkttaste_mittefahren:= ,
				b_direkttaste_einfahren	:= ,
				e_druckwaechter:= ST_Betriebsfreigaben.e_druckwaechter,
				i16_betriebsart:= gi16_betriebsart,
				b_no_gesteuert_im_norm_betrieb:= ,
				st_ctrl_in:= zyl_haspel_verschieben.st_ctrl.in,
				b_masterachse_hand_dialog_aktiv:= ,
				st_visu:= visu.st_zyl,
				st_ctrl_out=> zyl_haspel_verschieben.st_ctrl.out,
				a_ventil_einfahren=> ,
				a_ventil_ausfahren=> );

			zyl_bandeinzuege_verschieben.fb(
				st_config:= ,
				bw_nocken_zylinder_einfahren:= ,
				bw_nocken_zylinder_ausfahren:= ,
				uw_nocken_zylinder_einfahren:= ,
				uw_nocken_zylinder_ausfahren:= ,
				b_direkttaste_ausfahren:= ,
				b_direkttaste_mittefahren:= ,
				b_direkttaste_einfahren	:= ,
				e_druckwaechter:= ST_Betriebsfreigaben.e_druckwaechter,
				i16_betriebsart:= gi16_betriebsart,
				b_no_gesteuert_im_norm_betrieb:= ,
				st_ctrl_in:= zyl_bandeinzuege_verschieben.st_ctrl.in,
				b_masterachse_hand_dialog_aktiv:= ,
				st_visu:= visu.st_zyl,
				st_ctrl_out=> zyl_bandeinzuege_verschieben.st_ctrl.out,
				a_ventil_einfahren=> ,
				a_ventil_ausfahren=> );
	
			zyl_rafo_faenger.fb.st_config.b_aktiv := NOT gst_datensatz.st_md.b_wt_transport_simulation;
			zyl_rafo_faenger.fb(
				st_config:= ,
				bw_nocken_zylinder_einfahren:= ,
				bw_nocken_zylinder_ausfahren:= ,
				uw_nocken_zylinder_einfahren:= ,
				uw_nocken_zylinder_ausfahren:= ,
				b_direkttaste_ausfahren:= ,
				b_direkttaste_mittefahren:= ,
				b_direkttaste_einfahren	:= ,
				e_druckwaechter:= ST_Betriebsfreigaben.e_druckwaechter,
				i16_betriebsart:= gi16_betriebsart,
				b_no_gesteuert_im_norm_betrieb:= ,
				st_ctrl_in:= zyl_rafo_faenger.st_ctrl.in,
				b_masterachse_hand_dialog_aktiv:= ,
				st_visu:= visu.st_zyl,
				st_ctrl_out=> zyl_rafo_faenger.st_ctrl.out,
				a_ventil_einfahren=> a_zyl_faenger_einfahren,
				a_ventil_ausfahren=> );
	
			zyl_rafo_klemmen.fb.st_config.b_aktiv := NOT gst_datensatz.st_md.b_wt_transport_simulation;
			zyl_rafo_klemmen.fb(
				st_config:= ,
				bw_nocken_zylinder_einfahren:= ,
				bw_nocken_zylinder_ausfahren:= ,
				uw_nocken_zylinder_einfahren:= ,
				uw_nocken_zylinder_ausfahren:= ,
				b_direkttaste_ausfahren:= ,
				b_direkttaste_mittefahren:= ,
				b_direkttaste_einfahren	:= ,
				e_druckwaechter:= ST_Betriebsfreigaben.e_druckwaechter,
				i16_betriebsart:= gi16_betriebsart,
				b_no_gesteuert_im_norm_betrieb:= ,
				st_ctrl_in:= zyl_rafo_klemmen.st_ctrl.in,
				b_masterachse_hand_dialog_aktiv:= ,
				st_visu:= visu.st_zyl,
				st_ctrl_out=> zyl_rafo_klemmen.st_ctrl.out,
				a_ventil_einfahren=> a_zyl_klemmen_einfahren,
				a_ventil_ausfahren=> );
	
			zyl_rafo_vorschub.fb.st_config.b_aktiv := NOT gst_datensatz.st_md.b_wt_transport_simulation;
			zyl_rafo_vorschub.fb(
				st_config:= ,
				bw_nocken_zylinder_einfahren:= ,
				bw_nocken_zylinder_ausfahren:= ,
				uw_nocken_zylinder_einfahren:= ,
				uw_nocken_zylinder_ausfahren:= ,
				b_direkttaste_ausfahren:= ,
				b_direkttaste_mittefahren:= ,
				b_direkttaste_einfahren	:= ,
				e_druckwaechter:= ST_Betriebsfreigaben.e_druckwaechter,
				i16_betriebsart:= gi16_betriebsart,
				b_no_gesteuert_im_norm_betrieb:= ,
				st_ctrl_in:= zyl_rafo_vorschub.st_ctrl.in,
				b_masterachse_hand_dialog_aktiv:= ,
				st_visu:= visu.st_zyl,
				st_ctrl_out=> zyl_rafo_vorschub.st_ctrl.out,
				a_ventil_einfahren=> a_zyl_vorschub_einfahren,
				a_ventil_ausfahren=> a_zyl_vorschub_ausfahren);
	
			zyl_rafo_kamm.fb.st_config.b_aktiv := NOT gst_datensatz.st_md.b_wt_transport_simulation;
			zyl_rafo_kamm.fb(
				st_config:= ,
				bw_nocken_zylinder_einfahren:= ,
				bw_nocken_zylinder_ausfahren:= ,
				uw_nocken_zylinder_einfahren:= ,
				uw_nocken_zylinder_ausfahren:= ,
				b_direkttaste_ausfahren:= ,
				b_direkttaste_mittefahren:= ,
				b_direkttaste_einfahren	:= ,
				e_druckwaechter:= ST_Betriebsfreigaben.e_druckwaechter,
				i16_betriebsart:= gi16_betriebsart,
				b_no_gesteuert_im_norm_betrieb:= ,
				st_ctrl_in:= zyl_rafo_kamm.st_ctrl.in,
				b_masterachse_hand_dialog_aktiv:= ,
				st_visu:= visu.st_zyl,
				st_ctrl_out=> zyl_rafo_kamm.st_ctrl.out,
				a_ventil_einfahren=> ,
				a_ventil_ausfahren=> );
	
			zyl_rafo_vorzentrierer.fb.st_config.b_aktiv := NOT gst_datensatz.st_md.b_wt_transport_simulation;
			zyl_rafo_vorzentrierer.fb(
				st_config:= ,
				bw_nocken_zylinder_einfahren:= ,
				bw_nocken_zylinder_ausfahren:= ,
				uw_nocken_zylinder_einfahren:= ,
				uw_nocken_zylinder_ausfahren:= ,
				b_direkttaste_ausfahren:= ,
				b_direkttaste_mittefahren:= ,
				b_direkttaste_einfahren	:= ,
				e_druckwaechter:= ST_Betriebsfreigaben.e_druckwaechter,
				i16_betriebsart:= gi16_betriebsart,
				b_no_gesteuert_im_norm_betrieb:= ,
				st_ctrl_in:= zyl_rafo_vorzentrierer.st_ctrl.in,
				b_masterachse_hand_dialog_aktiv:= ,
				st_visu:= visu.st_zyl,
				st_ctrl_out=> zyl_rafo_vorzentrierer.st_ctrl.out,
				a_ventil_einfahren=> ,
				a_ventil_ausfahren=> );
	END_CASE
END_IF
END_PROGRAM

(* POU Gemeinsamkeiten17xx/Zylinder/ST_Zylinder_Fast, ST *)
PROGRAM ST_Zylinder_Fast
VAR
END_VAR
(* Zylinderaufrufe *)
CASE gst_datensatz.st_md.i16_typ_zelle OF
	KEINE_ZELLE:
		;

	BESTUECKZELLE_1700:
		ST_Datainit_Fast_Zylinder();

		CASE gst_datensatz.st_wkz.i16_typ_bandeinzug OF
			KEIN_EINZUG:
				;

			STANDARD_2FACH_V2:
				;

				BANDWECHSLER_V2:
				zyl_bandfaenger.fb.st_config.b_aktiv := NOT gst_datensatz.st_md.b_wt_transport_simulation;
				zyl_bandfaenger.fb(
					st_config:= ,
					e_druckwaechter:= ST_Betriebsfreigaben.e_druckwaechter,
					i16_betriebsart:= gi16_betriebsart,
					b_no_gesteuert_im_norm_betrieb:= ,
					b_direkttaste_ausfahren:= ,
					b_direkttaste_mittefahren:= ,
					b_direkttaste_einfahren	:= ,
					st_ctrl_in:= zyl_bandfaenger.st_ctrl.in,
					b_masterachse_hand_dialog_aktiv:= ST_Bestueckachse.b_hand_dialog_aktiv,
					st_visu:= visu.st_zyl,
					bw_nocken_zylinder_einfahren := nockenschaltwerk_bestueckachse.fb.arr_spur[SP_BW_BANDFAENGER_BAWEV2_EINFAHREN],
					bw_nocken_zylinder_ausfahren := nockenschaltwerk_bestueckachse.fb.arr_spur[SP_BW_BANDFAENGER_BAWEV2_AUSFAHREN],
					uw_nocken_zylinder_einfahren := ,
					uw_nocken_zylinder_ausfahren := ,
					st_ctrl_out=> zyl_bandfaenger.st_ctrl.out,
					a_ventil_einfahren=> a_zyl_faenger_einfahren,
					a_ventil_ausfahren=> );
		
				zyl_bandklemmen.fb.st_config.b_aktiv := NOT gst_datensatz.st_md.b_wt_transport_simulation;
				zyl_bandklemmen.fb(
					st_config:= ,
					e_druckwaechter:= ST_Betriebsfreigaben.e_druckwaechter,
					i16_betriebsart:= gi16_betriebsart,
					b_no_gesteuert_im_norm_betrieb:= ,
					b_direkttaste_ausfahren:= ,
					b_direkttaste_mittefahren:= ,
					b_direkttaste_einfahren	:= ,
					st_ctrl_in:= zyl_bandklemmen.st_ctrl.in,
					b_masterachse_hand_dialog_aktiv:= ST_Bestueckachse.b_hand_dialog_aktiv,
					st_visu:= visu.st_zyl,
					bw_nocken_zylinder_einfahren := nockenschaltwerk_bestueckachse.fb.arr_spur[SP_BW_BANDKLEMMEN_BAWEV2_EINFAHREN],
					bw_nocken_zylinder_ausfahren := nockenschaltwerk_bestueckachse.fb.arr_spur[SP_BW_BANDKLEMMEN_BAWEV2_AUSFAHREN],
					uw_nocken_zylinder_einfahren :=  ,
					uw_nocken_zylinder_ausfahren :=  ,
					st_ctrl_out=> zyl_bandklemmen.st_ctrl.out,
					a_ventil_einfahren=> a_zyl_klemmen_einfahren,
					a_ventil_ausfahren=> );

				IF NOT gst_datensatz.st_md.b_auswahlSpruehoeler THEN
					zyl_oelen_oben.fb(
						st_config:= ,
						e_druckwaechter:= ST_Betriebsfreigaben.e_druckwaechter,
						i16_betriebsart:= gi16_betriebsart,
						b_no_gesteuert_im_norm_betrieb:= ,
						b_direkttaste_ausfahren:= ,
						b_direkttaste_mittefahren:= ,
						b_direkttaste_einfahren	:= ,
						st_ctrl_in:=zyl_oelen_oben.st_ctrl.in ,
						b_masterachse_hand_dialog_aktiv:=ST_Bestueckachse.b_hand_dialog_aktiv,
						st_visu:= visu.st_zyl,
						bw_nocken_zylinder_einfahren := (*ST_BandoelerZylinder.b_zyl_oben = FALSE OR*) nockenschaltwerk_bestueckachse.fb.arr_spur[56],
						bw_nocken_zylinder_ausfahren := (*ST_BandoelerZylinder.b_zyl_oben = TRUE AND*)  nockenschaltwerk_bestueckachse.fb.arr_spur[57],
						uw_nocken_zylinder_einfahren := zyl_oelen_oben.fb.e_sensor1_eingefahren AND  nockenschaltwerk_bestueckachse.fb.arr_spur[58],
						uw_nocken_zylinder_ausfahren := zyl_oelen_oben.fb.e_sensor1_ausgefahren AND  nockenschaltwerk_bestueckachse.fb.arr_spur[59],
						st_ctrl_out=> zyl_oelen_oben.st_ctrl.out,
						a_ventil_einfahren=> ,
						a_ventil_ausfahren=> );
	
					gst_datensatz.st_wkz.nockenschaltwerk_bestueckachse.arr_nocken[56].b_camvalid := TRUE;
					gst_datensatz.st_wkz.nockenschaltwerk_bestueckachse.arr_nocken[57].b_camvalid := TRUE;
					gst_datensatz.st_wkz.nockenschaltwerk_bestueckachse.arr_nocken[58].b_camvalid := TRUE;
					gst_datensatz.st_wkz.nockenschaltwerk_bestueckachse.arr_nocken[59].b_camvalid := TRUE;
	
					zyl_oelen_unten.fb(
						st_config:= ,
						e_druckwaechter:= ST_Betriebsfreigaben.e_druckwaechter,
						i16_betriebsart:= gi16_betriebsart,
						b_no_gesteuert_im_norm_betrieb:= ,
						b_direkttaste_ausfahren:= ,
						b_direkttaste_mittefahren:= ,
						b_direkttaste_einfahren	:= ,
						st_ctrl_in:=zyl_oelen_unten.st_ctrl.in ,
						b_masterachse_hand_dialog_aktiv:=ST_Bestueckachse.b_hand_dialog_aktiv,
						st_visu:= visu.st_zyl,
						bw_nocken_zylinder_einfahren := nockenschaltwerk_bestueckachse.fb.arr_spur[60],
						bw_nocken_zylinder_ausfahren := nockenschaltwerk_bestueckachse.fb.arr_spur[61],
						uw_nocken_zylinder_einfahren := zyl_oelen_unten.fb.e_sensor1_eingefahren AND nockenschaltwerk_bestueckachse.fb.arr_spur[62],
						uw_nocken_zylinder_ausfahren := zyl_oelen_unten.fb.e_sensor1_ausgefahren AND  nockenschaltwerk_bestueckachse.fb.arr_spur[63],
						st_ctrl_out=>zyl_oelen_unten.st_ctrl.out ,
						a_ventil_einfahren=> ,
						a_ventil_ausfahren=> );
	
					gst_datensatz.st_wkz.nockenschaltwerk_bestueckachse.arr_nocken[60].b_camvalid := TRUE;
					gst_datensatz.st_wkz.nockenschaltwerk_bestueckachse.arr_nocken[61].b_camvalid := TRUE;
					gst_datensatz.st_wkz.nockenschaltwerk_bestueckachse.arr_nocken[62].b_camvalid := TRUE;
					gst_datensatz.st_wkz.nockenschaltwerk_bestueckachse.arr_nocken[63].b_camvalid := TRUE;
				END_IF

			SERVO:
				;
		END_CASE

	BESTUECKZELLE_1720:
		ST_Datainit_Fast_Zylinder();

		CASE gst_datensatz.st_wkz.i16_typ_bandeinzug OF
			KEIN_EINZUG:
				;
		
			STANDARD_2FACH_V2:
				zyl_bandfaenger_li.fb(
					st_config:= ,
					e_druckwaechter:= ST_Betriebsfreigaben.e_druckwaechter,
					i16_betriebsart:= gi16_betriebsart,
					b_no_gesteuert_im_norm_betrieb:= ,
					b_direkttaste_ausfahren:= ,
					b_direkttaste_mittefahren:= ,
					b_direkttaste_einfahren	:= ,
					st_ctrl_in:= zyl_bandfaenger_li.st_ctrl.in,
					b_masterachse_hand_dialog_aktiv:= ST_Bestueckachse.b_hand_dialog_aktiv,
					st_visu:= visu.st_zyl,
					bw_nocken_zylinder_einfahren := nockenschaltwerk_bestueckachse.fb.arr_spur[SP_BW_BANDFAENGER_LI_BAEZV2_EINFAHREN],
					bw_nocken_zylinder_ausfahren := nockenschaltwerk_bestueckachse.fb.arr_spur[SP_BW_BANDFAENGER_LI_BAEZV2_AUSFAHREN],
					uw_nocken_zylinder_einfahren := ,
					uw_nocken_zylinder_ausfahren := ,
					st_ctrl_out=> zyl_bandfaenger_li.st_ctrl.out,
					a_ventil_einfahren=> ,
					a_ventil_ausfahren=> );
				
				zyl_bandfaenger_re.fb(
					st_config:= ,
					e_druckwaechter:= ST_Betriebsfreigaben.e_druckwaechter,
					i16_betriebsart:= gi16_betriebsart,
					b_no_gesteuert_im_norm_betrieb:= ,
					b_direkttaste_ausfahren:= ,
					b_direkttaste_mittefahren:= ,
					b_direkttaste_einfahren	:= ,
					st_ctrl_in:= zyl_bandfaenger_re.st_ctrl.in,
					b_masterachse_hand_dialog_aktiv:= ST_Bestueckachse.b_hand_dialog_aktiv,
					st_visu:= visu.st_zyl,
					bw_nocken_zylinder_einfahren := nockenschaltwerk_bestueckachse.fb.arr_spur[SP_BW_BANDFAENGER_RE_BAEZV2_EINFAHREN],
					bw_nocken_zylinder_ausfahren := nockenschaltwerk_bestueckachse.fb.arr_spur[SP_BW_BANDFAENGER_RE_BAEZV2_AUSFAHREN],
					uw_nocken_zylinder_einfahren := ,
					uw_nocken_zylinder_ausfahren := ,
					st_ctrl_out=> zyl_bandfaenger_re.st_ctrl.out,
					a_ventil_einfahren=> ,
					a_ventil_ausfahren=> );
		
				zyl_bandklemmen_li.fb(
					st_config:= ,
					e_druckwaechter:= ST_Betriebsfreigaben.e_druckwaechter,
					i16_betriebsart:= gi16_betriebsart,
					b_no_gesteuert_im_norm_betrieb:= ,
					b_direkttaste_ausfahren:= ,
					b_direkttaste_mittefahren:= ,
					b_direkttaste_einfahren	:= ,
					st_ctrl_in:= zyl_bandklemmen_li.st_ctrl.in,
					b_masterachse_hand_dialog_aktiv:= ST_Bestueckachse.b_hand_dialog_aktiv,
					st_visu:= visu.st_zyl,
					bw_nocken_zylinder_einfahren := nockenschaltwerk_bestueckachse.fb.arr_spur[SP_BW_BANDKLEMMEN_LI_BAEZV2_EINFAHREN],
					bw_nocken_zylinder_ausfahren := nockenschaltwerk_bestueckachse.fb.arr_spur[SP_BW_BANDKLEMMEN_LI_BAEZV2_AUSFAHREN],
					uw_nocken_zylinder_einfahren := ,
					uw_nocken_zylinder_ausfahren := ,
					st_ctrl_out=> zyl_bandklemmen_li.st_ctrl.out,
					a_ventil_einfahren=> ,
					a_ventil_ausfahren=> );
				
				zyl_bandklemmen_re.fb(
					st_config:= ,
					e_druckwaechter:= ST_Betriebsfreigaben.e_druckwaechter,
					i16_betriebsart:= gi16_betriebsart,
					b_no_gesteuert_im_norm_betrieb:= ,
					b_direkttaste_ausfahren:= ,
					b_direkttaste_mittefahren:= ,
					b_direkttaste_einfahren	:= ,
					st_ctrl_in:= zyl_bandklemmen_re.st_ctrl.in,
					b_masterachse_hand_dialog_aktiv:= ST_Bestueckachse.b_hand_dialog_aktiv,
					st_visu:= visu.st_zyl,
					bw_nocken_zylinder_einfahren := nockenschaltwerk_bestueckachse.fb.arr_spur[SP_BW_BANDKLEMMEN_RE_BAEZV2_EINFAHREN],
					bw_nocken_zylinder_ausfahren := nockenschaltwerk_bestueckachse.fb.arr_spur[SP_BW_BANDKLEMMEN_RE_BAEZV2_AUSFAHREN],
					uw_nocken_zylinder_einfahren := ,
					uw_nocken_zylinder_ausfahren := ,
					st_ctrl_out=> zyl_bandklemmen_re.st_ctrl.out,
					a_ventil_einfahren=> ,
					a_ventil_ausfahren=> );

			BANDWECHSLER_V2:
				;

			SERVO:
				;
		END_CASE;

	RASTERFOLIE:
		;
END_CASE
END_PROGRAM

(* POU MAINs/MAIN_BBGen, ST *)
PROGRAM MAIN_BBGen
VAR
END_VAR
(* BBGen in einem extra Task um lange Berechnungen zu ermöglichen ohne dass die Verbindung zum Prozessabbild abbricht *)
(* Fehlermeldung sonst: Watchdog des asynchronen Mapping 5 zwischen Prozeßabbild 2 und 6 hat zugeschlagen, da Prozeßabbild 2 keine neuen Daten lieferte
 * Die Safty schaltet sonst alles ab *)


ST_BBGen(
	st_config:= bbgen.st_config,
	st_visu:= visu.st_xml_server,
	st_ctrl_in:= bbgen.st_ctrl.in,
	st_ctrl_out=> bbgen.st_ctrl.out,
	i16_auftrag:= gi16_bbgen_auftrag);


(*Maschinendaten müssen bereits ausgelesen sein.*)
IF gst_datensatz.st_md.i16_typ_zelle <> KEINE_ZELLE THEN
	ST_Wartung(
		st_config:= wartung.st_config,
		st_ctrl_in:= wartung.st_ctrl.in,
		st_ctrl_out=> wartung.st_ctrl.out,
		i16_auftrag:= gi16_wartung_auftrag);
END_IF
END_PROGRAM

(* POU MAINs/MAIN_FAST, ST *)
PROGRAM MAIN_FAST
VAR
END_VAR
CASE gst_datensatz.st_md.i16_typ_zelle OF
	KEINE_ZELLE:
		ST_Safetyprogramm(
			st_config:= safety.st_config,
			st_ctrl_in:= safety.st_ctrl.in,
			st_visu:= safety.st_visu,
			st_ctrl_out=> safety.st_ctrl.out);

		ST_Betriebsfreigaben(
			st_config:= betriebsfreigaben.st_config,
			st_ctrl_in:= betriebsfreigaben.st_ctrl.in,
			b_lampe_stoerung:= ,
			b_lampe_produktion:= ,
			e_steuerung_ein:= ST_Safetyprogramm.se_steuerung_ein,
			st_ctrl_out=> betriebsfreigaben.st_ctrl.out);

		nockenschaltwerk_bestueckachse.fb(
			r_achsposition:= virtuelle_master_achse.NcToPlc.ModuloActPos,
			r_achsgeschwindigkeit:= virtuelle_master_achse.NcToPlc.ActVelo * 60 / 360,
			i16_verfahrrichtung_achse_extern:=  ,
			b_verfahrrichtungsauswertung_extern:= FALSE,
			i16_art_der_achse:= RUND,
			st_config:= nockenschaltwerk_bestueckachse.st_config,
			arr_nocken:= gst_datensatz.st_wkz.nockenschaltwerk_bestueckachse.arr_nocken,
			st_visu:= visu);

	BESTUECKZELLE_1700:
		ST_Safetyprogramm(
			st_config:= safety.st_config,
			st_ctrl_in:= safety.st_ctrl.in,
			st_visu:= safety.st_visu,
			st_ctrl_out=> safety.st_ctrl.out);

		ST_Betriebsfreigaben(
			st_config:= betriebsfreigaben.st_config,
			st_ctrl_in:= betriebsfreigaben.st_ctrl.in,
			b_lampe_stoerung:= ,
			b_lampe_produktion:= ,
			e_steuerung_ein:= ST_Safetyprogramm.se_steuerung_ein,
			st_ctrl_out=> betriebsfreigaben.st_ctrl.out);

		nockenschaltwerk_bestueckachse.fb(
			r_achsposition:= virtuelle_master_achse.NcToPlc.ModuloActPos,
			r_achsgeschwindigkeit:= virtuelle_master_achse.NcToPlc.ActVelo * 60 / 360,
			i16_verfahrrichtung_achse_extern:=  ,
			b_verfahrrichtungsauswertung_extern:= FALSE,
			i16_art_der_achse:= RUND,
			st_config:= nockenschaltwerk_bestueckachse.st_config,
			arr_nocken:= gst_datensatz.st_wkz.nockenschaltwerk_bestueckachse.arr_nocken,
			st_visu:= visu);

		ST_Virtuelle_Masterachse(
			st_config_achse:= axis_virt_master.st_config,
			e_ls_bandende_re := ST_Bandwechsel_Kontroller.e_ls_bandende_re,
			e_ls_bandende_li	:= ST_Bandwechsel_Kontroller.e_ls_bandende_li,
			st_ctrl_in:= axis_virt_master.st_ctrl.in,
			e_steuerung_ein:= ST_Safetyprogramm.se_steuerung_ein,
			e_ba_mit_bedingungen:= ST_Safetyprogramm.se_ba_mit_bedingungen,
			st_visu:= axis_virt_master.st_visu,
			st_visu_virtuell:= axis_virt_master.st_visu,
			st_ctrl_out=> axis_virt_master.st_ctrl.out,
			b_materialmangel=> ST_LampeMaterialMangel.b_materialmangel[2],
			b_materialmangel2=> ST_LampeMaterialMangel.b_materialmangel[6]);

		CASE gst_datensatz.st_wkz.i16_typ_bandeinzug OF
			KEIN_EINZUG:
				;
			STANDARD_2FACH_V2:
				;
			BANDWECHSLER_V2:
				;
			SERVO:
				ST_Servobandeinzug(
					st_config_achse:= axis_bandeinzug_achse.st_config,
					st_ctrl_in:= axis_bandeinzug_achse.st_ctrl.in,
					e_steuerung_ein:= ST_Safetyprogramm.se_steuerung_ein,
					e_ba_mit_bedingungen:= ST_Safetyprogramm.se_ba_mit_bedingungen,
					e_tuere_vorne_offen:= ST_Safetyprogramm.se_tuere_vorne_offen,
					e_tuere_hinten_offen:= ST_Safetyprogramm.se_tuere_hinten_offen,
					st_visu:= axis_bandeinzug_achse.st_visu,
					st_ctrl_out=> axis_bandeinzug_achse.st_ctrl.out);
		END_CASE

		ST_WkzAbsicherung(
			st_config:= wkz_absicherung.st_config,
			st_ctrl_in:= wkz_absicherung.st_ctrl.in,
			st_visu:= wkz_absicherung.st_visu,
			st_ctrl_out=> wkz_absicherung.st_ctrl.out);

		ST_Einpress_Kontroller(
			st_config:= einpresskraft_kontroller.st_config,
			st_ctrl_in:= einpresskraft_kontroller.st_ctrl.in,
			lr_achsposition:= bestueckachse.NcToPlc.ModuloActPos,
			st_visu:= einpresskraft_kontroller.st_visu,
			st_einpressen:= gst_datensatz.st_band.st_einpressen,
			st_ctrl_out=> einpresskraft_kontroller.st_ctrl.out);


		ST_Bandeinzug_Kontroller_1700(
			st_config:= bandeinzug_kontroller.st_config,
			st_ctrl_in:= bandeinzug_kontroller.st_ctrl.in,
			st_visu:= bandeinzug_kontroller.st_visu,
			st_ctrl_out=> bandeinzug_kontroller.st_ctrl.out);

		ST_Zylinder_Fast();

	BESTUECKZELLE_1720:
		ST_Safetyprogramm(
			st_config:= safety.st_config,
			st_ctrl_in:= safety.st_ctrl.in,
			st_visu:= safety.st_visu,
			st_ctrl_out=> safety.st_ctrl.out);

		ST_Betriebsfreigaben(
			st_config:= betriebsfreigaben.st_config,
			st_ctrl_in:= betriebsfreigaben.st_ctrl.in,
			b_lampe_stoerung:= ,
			b_lampe_produktion:= ,
			e_steuerung_ein:= ST_Safetyprogramm.se_steuerung_ein,
			st_ctrl_out=> betriebsfreigaben.st_ctrl.out);
		
		nockenschaltwerk_bestueckachse.fb(
			r_achsposition:= virtuelle_master_achse.NcToPlc.ModuloActPos,
			r_achsgeschwindigkeit:= virtuelle_master_achse.NcToPlc.ActVelo * 60 / 360,
			i16_verfahrrichtung_achse_extern:=  ,
			b_verfahrrichtungsauswertung_extern:= FALSE,
			i16_art_der_achse:= RUND,
			st_config:= nockenschaltwerk_bestueckachse.st_config,
			arr_nocken:= gst_datensatz.st_wkz.nockenschaltwerk_bestueckachse.arr_nocken,
			st_visu:= visu);

		ST_Virtuelle_Masterachse(
			st_config_achse:= axis_virt_master.st_config,
			e_ls_bandende_re := ST_Bandeinzug_Kontroller_1720.e_ls_bandende_re,
			e_ls_bandende_li	:= ST_Bandeinzug_Kontroller_1720.e_ls_bandende_li,
			st_ctrl_in:= axis_virt_master.st_ctrl.in,
			e_steuerung_ein:= ST_Safetyprogramm.se_steuerung_ein,
			e_ba_mit_bedingungen:= ST_Safetyprogramm.se_ba_mit_bedingungen,
			st_visu:= axis_virt_master.st_visu,
			st_visu_virtuell:= axis_virt_master.st_visu,
			st_ctrl_out=> axis_virt_master.st_ctrl.out,
			b_materialmangel=> ST_LampeMaterialMangel.b_materialmangel[2],
			b_materialmangel2=> ST_LampeMaterialMangel.b_materialmangel[6]);

		ST_WkzAbsicherung(
			st_config:= wkz_absicherung.st_config,
			st_ctrl_in:= wkz_absicherung.st_ctrl.in,
			st_visu:= wkz_absicherung.st_visu,
			st_ctrl_out=> wkz_absicherung.st_ctrl.out);

		ST_Bandeinzug_Kontroller_1720(
			st_config:= bandeinzug_kontroller.st_config,
			st_ctrl_in:= bandeinzug_kontroller.st_ctrl.in,
			st_visu:= bandeinzug_kontroller.st_visu,
			st_ctrl_out=> bandeinzug_kontroller.st_ctrl.out);

		ST_Zylinder_Fast();

	RASTERFOLIE:
		ST_Safetyprogramm(
			st_config:= safety.st_config,
			st_ctrl_in:= safety.st_ctrl.in,
			st_visu:= safety.st_visu,
			st_ctrl_out=> safety.st_ctrl.out);
	
		ST_Betriebsfreigaben(
			st_config:= betriebsfreigaben.st_config,
			st_ctrl_in:= betriebsfreigaben.st_ctrl.in,
			b_lampe_stoerung:= ,
			b_lampe_produktion:= ,
			e_steuerung_ein:= ST_Safetyprogramm.se_steuerung_ein,
			st_ctrl_out=> betriebsfreigaben.st_ctrl.out);
		
		nockenschaltwerk_bestueckachse.fb(
			r_achsposition:= virtuelle_master_achse.NcToPlc.ModuloActPos,
			r_achsgeschwindigkeit:= virtuelle_master_achse.NcToPlc.ActVelo * 60 / 360,
			i16_verfahrrichtung_achse_extern:=  ,
			b_verfahrrichtungsauswertung_extern:= FALSE,
			i16_art_der_achse:= RUND,
			st_config:= nockenschaltwerk_bestueckachse.st_config,
			arr_nocken:= gst_datensatz.st_wkz.nockenschaltwerk_bestueckachse.arr_nocken,
			st_visu:= visu);

		ST_Virtuelle_Masterachse(
			st_config_achse:= axis_virt_master.st_config,
			e_ls_bandende_re := ST_Bandwechsel_Kontroller.e_ls_bandende_re,
			e_ls_bandende_li	:= ST_Bandwechsel_Kontroller.e_ls_bandende_li,
			st_ctrl_in:= axis_virt_master.st_ctrl.in,
			e_steuerung_ein:= ST_Safetyprogramm.se_steuerung_ein,
			e_ba_mit_bedingungen:= ST_Safetyprogramm.se_ba_mit_bedingungen,
			st_visu:= axis_virt_master.st_visu,
			st_visu_virtuell:= axis_virt_master.st_visu,
			st_ctrl_out=> axis_virt_master.st_ctrl.out,
			b_materialmangel=> ST_LampeMaterialMangel.b_materialmangel[2],
			b_materialmangel2=> ST_LampeMaterialMangel.b_materialmangel[6]);
END_CASE
END_PROGRAM

(* POU Maschine1700/Band/ST_Bandwechsel_Kontroller, ST *)
PROGRAM ST_Bandwechsel_Kontroller
VAR_INPUT
	st_config						: struct_config;
	st_ctrl_in						: struct_ctrl_in;
END_VAR
VAR_IN_OUT
	st_visu						: struct_visu;
END_VAR
VAR_OUTPUT
	st_ctrl_out					: struct_ctrl_out;
	b_materialmangel				: BOOL;
	b_materialmangel_links				: BOOL;
	b_materialmangel_rechts				: BOOL;
END_VAR
VAR
	fb_ton_wz					: TON;
	fb_ton_uez					: TON;
	fb_ton_quitt					: TON;
	fb_tof_bandende_li			: TOF;
	fb_tof_bandende_re			: TOF;
	fb_ton_bandende_li			: TON;
	fb_ton_bandende_re			: TON;
	fb_r_trig_start					: R_TRIG;
	fb_r_trig_auto_Bandwechsel_aus: R_TRIG;
	fb_state_entry					: ST_StateEntry;
	b_ibn_start					: BOOL := FALSE;
	fb_r_trig_ibn_start				: R_TRIG;
	fb_ton_ibn_start				: TON;
	i16_vorgabe_einfaedeln		: INT := 0;
	i16_akt_einfaedeln			: INT := 0;
	i16_vorgabe_ausfaedeln		: INT := 0;
	i16_akt_ausfaedeln			: INT := 0;
	i							: INT := 0;
	b_ausgefaedelt				: BOOL;
	b_spulenwechsel				: BOOL;

	sm_halter_nicht_oben			: BOOL:= FALSE;
	sm_bandwechsel_ohne_ende	: BOOL:= FALSE;
	sm_kein_band_anderer_einzug	: BOOL:= FALSE;
	sm_kein_band_in_akt_einzug	: BOOL:= FALSE;
	bm_bandwechselvorgang		: BOOL := FALSE;
	bm_bandwechsel_manuell		: BOOL := FALSE;

	e_ls_bandende_li				AT %I* : BOOL;
	e_ls_bandende_re			AT %I* : BOOL;
END_VAR
(* Zeiten *)
fb_ton_wz(IN:= , PT:= , Q=>  , ET=> );
fb_ton_uez(IN:= , PT:= , Q=>  , ET=> );
fb_ton_quitt(IN:= , PT:= t#100ms, Q=> , ET=> );

fb_ton_bandende_li(IN:= e_ls_bandende_li, PT:= t#1000ms, Q=> , ET=> );
fb_ton_bandende_re(IN:= e_ls_bandende_re, PT:= t#1000ms, Q=> , ET=> );
fb_tof_bandende_li(IN:= fb_ton_bandende_li.Q, PT:= t#1100ms, Q=> , ET=> );
fb_tof_bandende_re(IN:= fb_ton_bandende_re.Q, PT:= t#1100ms, Q=> , ET=> );

(* Flanken *)
fb_r_trig_start(CLK:= st_ctrl_in.b_start, Q=> );

(* Inbetriebnahme *)
fb_r_trig_ibn_start (CLK:= b_ibn_start , Q=> );
fb_ton_ibn_start (IN:= , PT:= t#1s, Q=> , ET=> );

IF fb_r_trig_ibn_start .Q THEN
	fb_ton_ibn_start .IN := TRUE;
ELSE
	IF fb_ton_ibn_start .Q THEN
		b_ibn_start  := FALSE;
	 	fb_ton_ibn_start .IN := FALSE;
	END_IF
END_IF

(* auto Bandwechsel aus *)
fb_r_trig_auto_Bandwechsel_aus(CLK:=visu_hinten.out.auto_Bandwechsel_aus, Q=>);

IF	fb_r_trig_auto_Bandwechsel_aus.Q THEN
	gst_datensatz.st_md.b_auto_Bandwechsel:=NOT gst_datensatz.st_md.b_auto_Bandwechsel;
END_IF
visu_hinten.in.Lampe_auto_Bandwechsel:=gst_datensatz.st_md.b_auto_Bandwechsel;


(* Hier nur Abschaltungen welche zum Bandwechsel Stop führen müssen *)
IF	axis_bestueckachse.st_ctrl.out.b_fehler OR
	axis_z_achse.st_ctrl.out.b_fehler OR
	axis_y_achse.st_ctrl.out.b_fehler OR
	bandspruehoeler.st_ctrl.out.b_fehler OR
	bandeinzug_kontroller.st_ctrl.out.b_fehler OR
	bandwechsel_kontroller.st_ctrl.out.b_fehler OR
	wkz_absicherung.st_ctrl.out.b_fehler OR
	wt_transport_kontroller.st_ctrl.out.b_fehler OR
	hublift_links.st_ctrl.out.b_fehler OR
	hublift_rechts.st_ctrl.out.b_fehler OR
	balluff_tag_reader.st_ctrl.out.b_fehler OR
	haspel_kontroller.st_ctrl.out.b_fehler OR
	bbgen.st_ctrl.out.b_fehler OR
	einpresskraft_kontroller.st_ctrl.out.b_fehler OR
	edit_mfps.st_ctrl.out.b_fehler OR
	Lesen_Schreiben_Tag.st_ctrl.out.b_fehler OR
	Service.st_ctrl.out.b_fehler OR
	gi16_betriebsart = HAND
	THEN
		visu_hinten.in.b_bandwechsel_aktiv := FALSE;
		visu_hinten.in.current_visu_folie := 'BA_1700_BAND_EINFAEDELN';
END_IF

(* Toplevel *)
IF fb_state_entry.i16_step < FEHLER THEN
	IF st_ctrl_in.b_stop THEN
		fb_state_entry.i16_next_step := STOP;
	END_IF
	(* Allgemeine Fehler *)
	IF	NOT gst_datensatz.st_md.b_wt_transport_simulation AND
		(zyl_bawe_vorschub.st_ctrl.out.b_fehler OR
		zyl_bawe_querschub.st_ctrl.out.b_fehler OR
		zyl_bawe_faenger_li.st_ctrl.out.b_fehler OR
		zyl_bawe_faenger_re.st_ctrl.out.b_fehler OR
		zyl_bawe_halter_li.st_ctrl.out.b_fehler OR
		zyl_bawe_halter_re.st_ctrl.out.b_fehler OR
		zyl_haspel_verschieben.st_ctrl.out.b_fehler OR
		zyl_bandeinzuege_verschieben.st_ctrl.out.b_fehler)
		THEN
			fb_state_entry.i16_next_step := FEHLER;
	(* Zylinder im Handbetrieb *)
	ELSIF gi16_betriebsart = HAND AND (
			(st_visu.st_zyl.i16_nr_zyl_im_handbetrieb = zyl_bawe_vorschub.fb.st_config.i16_identnummer) OR
			(st_visu.st_zyl.i16_nr_zyl_im_handbetrieb = zyl_bawe_querschub.fb.st_config.i16_identnummer) OR
			(st_visu.st_zyl.i16_nr_zyl_im_handbetrieb = zyl_bawe_faenger_li.fb.st_config.i16_identnummer) OR
			(st_visu.st_zyl.i16_nr_zyl_im_handbetrieb = zyl_bawe_faenger_re.fb.st_config.i16_identnummer ) OR
			(st_visu.st_zyl.i16_nr_zyl_im_handbetrieb = zyl_bawe_halter_li.fb.st_config.i16_identnummer) OR
			(st_visu.st_zyl.i16_nr_zyl_im_handbetrieb = zyl_bawe_halter_re.fb.st_config.i16_identnummer)OR
			(st_visu.st_zyl.i16_nr_zyl_im_handbetrieb = zyl_haspel_verschieben.fb.st_config.i16_identnummer)OR
			(st_visu.st_zyl.i16_nr_zyl_im_handbetrieb = zyl_bandeinzuege_verschieben.fb.st_config.i16_identnummer))
			THEN
				fb_state_entry.i16_next_step := FEHLER;
	END_IF
END_IF

(* Bandwechsel wird durch eine gelbe Dauerleuchte angezeigt *)
b_materialmangel := b_materialmangel_links OR b_materialmangel_rechts;

IF	b_ausgefaedelt THEN
	IF 	b_materialmangel_links AND
		NOT fb_tof_bandende_li.Q THEN
		b_materialmangel_links := FALSE;
		b_ausgefaedelt:=FALSE;
	END_IF
	IF 	b_materialmangel_rechts AND
		NOT fb_tof_bandende_re.Q   THEN
		b_materialmangel_rechts := FALSE;
		b_ausgefaedelt:=FALSE;
	END_IF
ELSE
	IF	gi16_maschinenstatusinfo = STATUS_MASCHINE_ARBEITET THEN
		IF 	NOT fb_tof_bandende_li.Q  AND zyl_bawe_querschub.fb.e_sensor1_eingefahren THEN
			b_materialmangel_links := TRUE;
		END_IF
		IF	NOT fb_tof_bandende_re.Q  AND zyl_bawe_querschub.fb.e_sensor1_ausgefahren THEN
			b_materialmangel_rechts := TRUE;
		END_IF
	END_IF
END_IF

(* ======================================Schrittkette======================================== *)
fb_state_entry(
	i16_next_step:= , 
	i16_pos:= 1,
	s_debugtext:= ,
	E=> ,
	X=> ,
	i16_step=> ,
	i16_last_step=> );

CASE fb_state_entry.i16_step OF
(*=======================================================*)
	INIT_OBJ:
		IF st_config.b_config_fertig THEN
			fb_state_entry.i16_next_step := INIT;
		END_IF

(*=======================================================*)
	INIT:
		IF fb_state_entry.E THEN
			fb_ton_wz.IN := FALSE;
			fb_ton_uez.IN	:= FALSE;
			fb_ton_quitt.IN := FALSE;
			sm_halter_nicht_oben := FALSE;
			sm_bandwechsel_ohne_ende := FALSE;
			sm_kein_band_anderer_einzug := FALSE;
			sm_kein_band_in_akt_einzug := FALSE;
			bm_bandwechselvorgang := FALSE;
			bm_bandwechsel_manuell := FALSE;
			st_ctrl_out.b_fehler := FALSE;
			st_ctrl_out.b_bereit := FALSE;
			st_ctrl_out.b_fertig := FALSE;
			st_ctrl_out.b_fertig_2 := FALSE;
			i16_vorgabe_ausfaedeln := 5;
			zyl_bawe_vorschub.st_ctrl.in.b_einfahren := FALSE;
			zyl_bawe_vorschub.st_ctrl.in.b_ausfahren := FALSE;
			zyl_bawe_querschub.st_ctrl.in.b_einfahren := FALSE;
			zyl_bawe_querschub.st_ctrl.in.b_ausfahren := FALSE;
			zyl_bawe_faenger_li.st_ctrl.in.b_einfahren := FALSE;
			zyl_bawe_faenger_li.st_ctrl.in.b_ausfahren := FALSE;
			zyl_bawe_faenger_re.st_ctrl.in.b_einfahren := FALSE;
			zyl_bawe_faenger_re.st_ctrl.in.b_ausfahren := FALSE;
			zyl_bawe_halter_li.st_ctrl.in.b_einfahren := FALSE;
			zyl_bawe_halter_li.st_ctrl.in.b_ausfahren := FALSE;
			zyl_bawe_halter_re.st_ctrl.in.b_einfahren := FALSE;
			zyl_bawe_halter_re.st_ctrl.in.b_ausfahren := FALSE;
			zyl_haspel_verschieben.st_ctrl.in.b_einfahren := FALSE;
			zyl_haspel_verschieben.st_ctrl.in.b_ausfahren := FALSE;
			zyl_bandeinzuege_verschieben.st_ctrl.in.b_einfahren := FALSE;
			zyl_bandeinzuege_verschieben.st_ctrl.in.b_ausfahren := FALSE;
			axis_bandeinzug_achse.st_ctrl.in.b_startpos := FALSE;
			visu_hinten.in.b_bandwechsel_aktiv := FALSE;
			b_materialmangel_links := FALSE;
			b_materialmangel_rechts := FALSE;
			b_ausgefaedelt:=FALSE;
			b_spulenwechsel:=FALSE;

			IF gst_datensatz.st_wkz.i16_typ_bandeinzug = SERVO THEN
				i16_vorgabe_einfaedeln :=2;
			ELSE
				i16_vorgabe_einfaedeln := gst_datensatz.st_wkz.i16_vorgabe_einfaedeln;
			END_IF
		END_IF

		(*-----------------------Weiterschaltbedingungen----------------------------*)
		IF st_ctrl_in.b_init THEN
			zyl_bawe_vorschub.st_ctrl.in.b_quittieren := FALSE;
			zyl_bawe_querschub.st_ctrl.in.b_quittieren := FALSE;
			zyl_bawe_faenger_li.st_ctrl.in.b_quittieren := FALSE;
			zyl_bawe_faenger_re.st_ctrl.in.b_quittieren := FALSE;
			zyl_bawe_halter_li.st_ctrl.in.b_quittieren := FALSE;
			zyl_bawe_halter_re.st_ctrl.in.b_quittieren := FALSE;
			zyl_haspel_verschieben.st_ctrl.in.b_quittieren := FALSE;
			zyl_bandeinzuege_verschieben.st_ctrl.in.b_quittieren := FALSE;

			IF NOT gst_datensatz.st_md.b_wt_transport_simulation THEN
				fb_state_entry.i16_next_step := 20;
			ELSE
				fb_state_entry.i16_next_step := BEREIT;
			END_IF
		END_IF

(*=======================================================*)
	20:	(* Abfrage Stellung Bandwechselquerschub  *)

		(*-----------------------Weiterschaltbedingungen----------------------------*)
		IF zyl_bawe_querschub.fb.e_sensor1_eingefahren THEN
			fb_state_entry.i16_next_step := 30;
		ELSIF zyl_bawe_querschub.fb.e_sensor1_ausgefahren THEN
			fb_state_entry.i16_next_step := 60;
		ELSE
			fb_state_entry.i16_next_step := 30;
		END_IF

(*=======================================================*)
	30:	(* Bandwechselquerschub einfahren *)
		IF fb_state_entry.E THEN
			zyl_bawe_querschub.st_ctrl.in.b_einfahren := TRUE;
		END_IF

		(*-----------------------Weiterschaltbedingungen----------------------------*)
		IF zyl_bawe_querschub.st_ctrl.out.b_eingefahren THEN
			zyl_bawe_querschub.st_ctrl.in.b_einfahren := FALSE;
			fb_state_entry.i16_next_step := 40;
		END_IF

(*=======================================================*)
	40:	(* Haspeln rechts: Haspel verschieben einfahren und Bandabzug ausfahren *)
		IF fb_state_entry.E THEN
			zyl_haspel_verschieben.st_ctrl.in.b_einfahren := TRUE;
			zyl_bandeinzuege_verschieben.st_ctrl.in.b_ausfahren := TRUE;
		END_IF
		(*-----------------------Weiterschaltbedingungen----------------------------*)
		IF  	zyl_haspel_verschieben.st_ctrl.out.b_eingefahren AND
 			zyl_bandeinzuege_verschieben.st_ctrl.out.b_ausgefahren
			THEN
				zyl_haspel_verschieben.st_ctrl.in.b_einfahren := FALSE;
				zyl_bandeinzuege_verschieben.st_ctrl.in.b_ausfahren := FALSE;
				fb_state_entry.i16_next_step := 50;
		END_IF

(*=======================================================*)
	50:	(* Halter rechts ausfahren und Band heben, Halter links einfahren  *)
		IF fb_state_entry.E THEN
			zyl_bawe_halter_re.st_ctrl.in.b_ausfahren := TRUE;
			zyl_bawe_halter_li.st_ctrl.in.b_einfahren := TRUE;
		END_IF

		(*-----------------------Weiterschaltbedingungen----------------------------*)
		IF 	zyl_bawe_halter_re.st_ctrl.out.b_ausgefahren AND
			zyl_bawe_halter_li.st_ctrl.out.b_eingefahren
			THEN
				zyl_bawe_halter_re.st_ctrl.in.b_ausfahren := FALSE;
				zyl_bawe_halter_li.st_ctrl.in.b_einfahren := FALSE;
				fb_state_entry.i16_next_step := 90;
		END_IF

(*=======================================================*)
	60:	(* Bandwechselquerschub ausfahren *)
		IF fb_state_entry.E THEN
			zyl_bawe_querschub.st_ctrl.in.b_ausfahren := TRUE;
		END_IF

		(*-----------------------Weiterschaltbedingungen----------------------------*)
		IF zyl_bawe_querschub.st_ctrl.out.b_ausgefahren THEN
			zyl_bawe_querschub.st_ctrl.in.b_ausfahren := FALSE;
			fb_state_entry.i16_next_step := 70;
		END_IF

(*=======================================================*)
	70:	(* Haspeln links: Haspel verschieben ausfahren und Bandabzug einfahren *)
		IF fb_state_entry.E THEN
			zyl_haspel_verschieben.st_ctrl.in.b_ausfahren := TRUE;
			zyl_bandeinzuege_verschieben.st_ctrl.in.b_einfahren := TRUE;
		END_IF
		(*-----------------------Weiterschaltbedingungen----------------------------*)
		IF  	zyl_haspel_verschieben.st_ctrl.out.b_ausgefahren AND
 			zyl_bandeinzuege_verschieben.st_ctrl.out.b_eingefahren
			THEN
				zyl_haspel_verschieben.st_ctrl.in.b_ausfahren := FALSE;
				zyl_bandeinzuege_verschieben.st_ctrl.in.b_einfahren := FALSE;
				fb_state_entry.i16_next_step := 80;
		END_IF

(*=======================================================*)
	80:	(* Halter links ausfahren und Band heben, Halter rechts einfahren  *)
		IF fb_state_entry.E THEN
			zyl_bawe_halter_li.st_ctrl.in.b_ausfahren := TRUE;
			zyl_bawe_halter_re.st_ctrl.in.b_einfahren := TRUE;
		END_IF

		(*-----------------------Weiterschaltbedingungen----------------------------*)
		IF 	zyl_bawe_halter_li.st_ctrl.out.b_ausgefahren AND
			zyl_bawe_halter_re.st_ctrl.out.b_eingefahren
			THEN
				zyl_bawe_halter_li.st_ctrl.in.b_ausfahren := FALSE;
				zyl_bawe_halter_re.st_ctrl.in.b_einfahren := FALSE;
				fb_state_entry.i16_next_step := 90;
		END_IF

(*=======================================================*)
	90:	(* Fänger links und rechts einfahren, damit Vorschub nach vorne fahren kann *)
		IF fb_state_entry.E THEN
			zyl_bawe_faenger_li.st_ctrl.in.b_einfahren := TRUE;
			zyl_bawe_faenger_re.st_ctrl.in.b_einfahren := TRUE;
		END_IF

		(*-----------------------Weiterschaltbedingungen----------------------------*)
		IF 	zyl_bawe_faenger_li.st_ctrl.out.b_eingefahren AND
			zyl_bawe_faenger_re.st_ctrl.out.b_eingefahren
			THEN
				zyl_bawe_faenger_li.st_ctrl.in.b_einfahren := FALSE;
				zyl_bawe_faenger_re.st_ctrl.in.b_einfahren := FALSE;
				fb_state_entry.i16_next_step := 95;
		END_IF

(*=======================================================*)
	95:	(* Vorschub ausfahren *)
		IF fb_state_entry.E THEN
			zyl_bawe_vorschub.st_ctrl.in.b_ausfahren := TRUE;
		END_IF

		(*-----------------------Weiterschaltbedingungen----------------------------*)
		IF zyl_bawe_vorschub.st_ctrl.out.b_ausgefahren THEN
			zyl_bawe_vorschub.st_ctrl.in.b_ausfahren := FALSE;
			fb_state_entry.i16_next_step := BEREIT;
		END_IF

(*=======================================================*)
	BEREIT:
		IF fb_state_entry.E THEN
			st_ctrl_out.b_bereit := TRUE;
			i16_akt_einfaedeln := 0;
			i16_akt_ausfaedeln := 0;
			bm_bandwechselvorgang := FALSE;
		END_IF

		(*-----------------------Weiterschaltbedingungen----------------------------*)
		(* Warte darauf, das ein Band leer wird und Starte Teil 1 zum Bandausfädeln *)
		(* Freigaben bei installietem Barcodereader wieder rein *)
		IF fb_r_trig_start.Q OR fb_r_trig_ibn_start.Q THEN
			st_ctrl_out.b_fertig := FALSE;
			st_ctrl_out.b_fertig_2 := FALSE;
			(* Nach dem Bandwechsel soll die Maschine in Einzelfertigung gehen*)
			IF NOT fb_tof_bandende_li.Q  AND zyl_bawe_querschub.fb.e_sensor1_eingefahren (*AND gst_barcode_persistent.b_band_rechts_ok*) THEN
				bm_bandwechselvorgang := TRUE;
				(* Nach dem Bandwechsel geht die Maschine in Abhängigkeit der Bedienereinstellung auf der Visu in Einzelfertigung *)
				fb_state_entry.i16_next_step := 200;
			ELSIF NOT fb_tof_bandende_re.Q  AND zyl_bawe_querschub.fb.e_sensor1_ausgefahren (* AND gst_barcode_persistent.b_band_links_ok*) THEN
				bm_bandwechselvorgang := TRUE;
				(* Nach dem Bandwechsel geht die Maschine in Abhängigkeit der Bedienereinstellung auf der Visu in Einzelfertigung *)
				fb_state_entry.i16_next_step := 500;
			ELSE
				sm_bandwechsel_ohne_ende := TRUE;
				fb_state_entry.i16_next_step := FEHLER;
			END_IF
		END_IF


(*---------------------------------------------------------------------------------------------------------------------------------------------------------------------------------------------------*)
(*========================Bandeinzug links ist leer===============================*)
	200:	(* Fänger links ausfahren zum Band halten, Fänger rechts einfahren zur Bandfreigabe im rechten Einzug - Halter gegensinnig *)
		IF fb_state_entry.E THEN
			zyl_bawe_faenger_li.st_ctrl.in.b_ausfahren := TRUE;
			zyl_bawe_faenger_re.st_ctrl.in.b_einfahren := TRUE;
			zyl_bawe_halter_li.st_ctrl.in.b_einfahren := TRUE;
			zyl_bawe_halter_re.st_ctrl.in.b_ausfahren := TRUE;
		END_IF

		(*-----------------------Weiterschaltbedingungen----------------------------*)
		IF 	zyl_bawe_faenger_li.st_ctrl.out.b_ausgefahren AND
			zyl_bawe_faenger_re.st_ctrl.out.b_eingefahren AND
			zyl_bawe_halter_li.st_ctrl.out.b_eingefahren AND
			zyl_bawe_halter_re.st_ctrl.out.b_ausgefahren AND
			gb_ba_auto_kontroller
			THEN
				zyl_bawe_faenger_li.st_ctrl.in.b_ausfahren := FALSE;
				zyl_bawe_faenger_re.st_ctrl.in.b_einfahren := FALSE;
				zyl_bawe_halter_li.st_ctrl.in.b_einfahren := FALSE;
				zyl_bawe_halter_re.st_ctrl.in.b_ausfahren := FALSE;
				fb_state_entry.i16_next_step := 210;
		END_IF

(*=======================================================*)
	210:	(* Band-Zylinder einfahren bzw. Servobandeinzug lösen *)
		CASE gst_datensatz.st_wkz.i16_typ_bandeinzug OF

			BANDWECHSLER_V2:
				IF fb_state_entry.E THEN
					(* Zylinder einfahren *)
					zyl_bandfaenger.st_ctrl.in.b_einfahren := TRUE;
					zyl_bandklemmen.st_ctrl.in.b_einfahren := TRUE;
				END_IF
					(* Bandwechsler V2 ohne Sensoren und anderen Zylindern *)
					gst_datensatz.st_wkz.nockenschaltwerk_bestueckachse.arr_nocken[NO_BW_BANDFAENGER_BAWEV2_EINFAHREN].b_camvalid := FALSE;
					gst_datensatz.st_wkz.nockenschaltwerk_bestueckachse.arr_nocken[NO_BW_BANDFAENGER_BAWEV2_AUSFAHREN].b_camvalid := FALSE;
					gst_datensatz.st_wkz.nockenschaltwerk_bestueckachse.arr_nocken[NO_BW_BANDKLEMMEN_BAWEV2_EINFAHREN].b_camvalid := FALSE;
					gst_datensatz.st_wkz.nockenschaltwerk_bestueckachse.arr_nocken[NO_BW_BANDKLEMMEN_BAWEV2_AUSFAHREN].b_camvalid := FALSE;
				(*-----------------------Weiterschaltbedingungen----------------------------*)
				IF 	zyl_bandfaenger.st_ctrl.out.b_eingefahren AND
					zyl_bandklemmen.st_ctrl.out.b_eingefahren AND
					gb_ba_auto_kontroller
					THEN
						zyl_bandfaenger.st_ctrl.in.b_einfahren := FALSE;
						zyl_bandklemmen.st_ctrl.in.b_einfahren := FALSE;
						fb_state_entry.i16_next_step := 220;
				END_IF

			SERVO:
				zyl_bawe_faenger_li.st_ctrl.in.b_einfahren := TRUE;
				zyl_bawe_halter_li.st_ctrl.in.b_einfahren := TRUE;
				(*-----------------------Weiterschaltbedingungen----------------------------*)
				IF 	zyl_bawe_faenger_li.st_ctrl.out.b_eingefahren AND
					zyl_bawe_halter_li.st_ctrl.out.b_eingefahren AND
					gb_ba_auto_kontroller
					THEN
						zyl_bawe_faenger_li.st_ctrl.in.b_einfahren := FALSE;
						zyl_bawe_halter_li.st_ctrl.in.b_einfahren := FALSE;
						fb_state_entry.i16_next_step := 216;
				END_IF
		END_CASE;

(*=======================================================*)
	216:	(* Servobandeinzug rückwärts fahren, damit die Ausschiebezylinder das Band sicher erwischen *)
		IF fb_state_entry.E THEN
			axis_bandeinzug_achse.st_ctrl.in.b_ausfaedeln_servo := TRUE;
		END_IF

		(*-----------------------Weiterschaltbedingungen----------------------------*)
		IF axis_bandeinzug_achse.st_ctrl.out.b_ausgefaedelt_servo AND NOT fb_state_entry.E THEN
			axis_bandeinzug_achse.st_ctrl.in.b_ausfaedeln_servo := FALSE;
			fb_state_entry.i16_next_step := 217;(*Neu*)
		END_IF

(*=======================================================*)
	217:	(* Fänger ins Band fahren, damit die Bremse gelöst werden kann *)
		IF fb_state_entry.E THEN
				zyl_bawe_faenger_li.st_ctrl.in.b_ausfahren := TRUE;
		END_IF

		(*-----------------------Weiterschaltbedingungen----------------------------*)
		IF 	zyl_bawe_faenger_li.st_ctrl.out.b_ausgefahren AND
			gb_ba_auto_kontroller
			THEN
				zyl_bawe_faenger_li.st_ctrl.in.b_ausfahren := FALSE;
				fb_state_entry.i16_next_step := 218;
		END_IF

(*=======================================================*)
	218:	(* Bremse an Servobandeinzug lösen, damit Band heraus gezogen werden kann. Die Bestückachse hat die Slavekopplung bereits gelöst. *)
		IF fb_state_entry.E THEN
			axis_bandeinzug_achse.st_ctrl.in.b_bremse_auf := TRUE;
		END_IF

		(*-----------------------Weiterschaltbedingungen----------------------------*)
		IF axis_bandeinzug_achse.st_ctrl.out.b_bremse_geoeffnet AND NOT fb_state_entry.E THEN
			axis_bandeinzug_achse.st_ctrl.in.b_bremse_auf := FALSE;
			fb_state_entry.i16_next_step := 220;
		END_IF

(*=======================================================*)
	220:	(* Vorschub einfahren und Band aus WKZ rausziehen *)
		IF fb_state_entry.E THEN
			zyl_bawe_vorschub.st_ctrl.in.b_einfahren := TRUE;
			i16_akt_ausfaedeln := i16_akt_ausfaedeln + 1;
		END_IF

		(*-----------------------Weiterschaltbedingungen----------------------------*)
		IF zyl_bawe_vorschub.st_ctrl.out.b_eingefahren AND gb_ba_auto_kontroller THEN
			zyl_bawe_vorschub.st_ctrl.in.b_einfahren := FALSE;
			IF i16_akt_ausfaedeln <= i16_vorgabe_ausfaedeln THEN
				fb_state_entry.i16_next_step := 230;
			ELSE
				fb_state_entry.i16_next_step := 280;
			END_IF
		END_IF

(*=======================================================*)
	230:	(* Bandwechselhalter links ausfahren um Band nachfassen zu können *)
		IF fb_state_entry.E THEN
			zyl_bawe_halter_li.st_ctrl.in.b_ausfahren := TRUE;
		END_IF

		(*-----------------------Weiterschaltbedingungen----------------------------*)
		IF zyl_bawe_halter_li.st_ctrl.out.b_ausgefahren AND gb_ba_auto_kontroller THEN
			zyl_bawe_halter_li.st_ctrl.in.b_ausfahren := FALSE;
			fb_state_entry.i16_next_step := 240;
		END_IF

(*=======================================================*)
	240:	(* Bandwechselfänger links einfahren*)
		IF fb_state_entry.E THEN
			zyl_bawe_faenger_li.st_ctrl.in.b_einfahren := TRUE;
		END_IF

		(*-----------------------Weiterschaltbedingungen----------------------------*)
		IF zyl_bawe_faenger_li.st_ctrl.out.b_eingefahren AND gb_ba_auto_kontroller THEN
			zyl_bawe_faenger_li.st_ctrl.in.b_einfahren := FALSE;
			fb_state_entry.i16_next_step := 250;
		END_IF

(*=======================================================*)
	250:	(* Vorschub ausfahren und Band nachfassen *)
		IF fb_state_entry.E THEN
			zyl_bawe_vorschub.st_ctrl.in.b_ausfahren := TRUE;
		END_IF

		(*-----------------------Weiterschaltbedingungen----------------------------*)
		IF zyl_bawe_vorschub.st_ctrl.out.b_ausgefahren AND gb_ba_auto_kontroller THEN
			zyl_bawe_vorschub.st_ctrl.in.b_ausfahren := FALSE;
			fb_state_entry.i16_next_step := 260;
		END_IF

(*=======================================================*)
	260:	(* Bandwechselfänger links ausfahren zum Band halten *)
		IF fb_state_entry.E THEN
			zyl_bawe_faenger_li.st_ctrl.in.b_ausfahren := TRUE;
		END_IF

		(*-----------------------Weiterschaltbedingungen----------------------------*)
		IF zyl_bawe_faenger_li.st_ctrl.out.b_ausgefahren AND gb_ba_auto_kontroller THEN
			zyl_bawe_faenger_li.st_ctrl.in.b_ausfahren := FALSE;
			fb_state_entry.i16_next_step := 270;
		END_IF

(*=======================================================*)
	270:	(* Bandwechselhalter links einfahren und Band freigeben*)
		IF fb_state_entry.E THEN
			zyl_bawe_halter_li.st_ctrl.in.b_einfahren := TRUE;
		END_IF

		(*-----------------------Weiterschaltbedingungen----------------------------*)
		IF zyl_bawe_halter_li.st_ctrl.out.b_eingefahren AND gb_ba_auto_kontroller THEN
			zyl_bawe_halter_li.st_ctrl.in.b_einfahren := FALSE;
			fb_state_entry.i16_next_step := 220;
		END_IF

(*=======================================================*)
	280:	(* Fänger links einfahren zum Ausfädeln *)
		IF fb_state_entry.E THEN
			zyl_bawe_faenger_li.st_ctrl.in.b_einfahren := TRUE;
		END_IF

		(*-----------------------Weiterschaltbedingungen----------------------------*)
		IF zyl_bawe_faenger_li.st_ctrl.out.b_eingefahren AND gb_ba_auto_kontroller THEN
			zyl_bawe_faenger_li.st_ctrl.in.b_einfahren := FALSE;
			fb_state_entry.i16_next_step := 290;
		END_IF

(*=======================================================*)
	290:	(* Band ist herausgezogen - prüfe Einstellung bzw. Bandanwesenheit im rechten Einzug *)
		b_ausgefaedelt:=b_materialmangel;
			(* Band vorhanden -> Beginn automatischer Bandwechsel *)
		(*-----------------------Weiterschaltbedingungen----------------------------*)
		IF fb_tof_bandende_re.Q AND gst_datensatz.st_md.b_auto_Bandwechsel THEN
			b_spulenwechsel := TRUE;
			fb_state_entry.i16_next_step := 300;
		ELSE
			(* Bandherausziehen ist fertig *)
			fb_state_entry.i16_next_step := 295;
		END_IF

(*=======================================================*)
	291:	(* Bediener muss am Backpanel auswählen ob Bandwechsel oder Trennstelle *)

		(*-----------------------Weiterschaltbedingungen----------------------------*)
		IF visu_hinten.out.b_Bandwechsel THEN
			(* Band vorhanden -> Beginn automatischer Bandwechsel *)
			visu_hinten.in.b_bandwechsel_aktiv := FALSE;
			visu_hinten.in.current_visu_folie := 'BESTUECKZELLE_1700';
			fb_state_entry.i16_next_step := 300;
		ELSIF visu_hinten.out.b_Trennstelle THEN
			visu_hinten.in.b_bandwechsel_aktiv := FALSE;
			CASE gst_datensatz.st_wkz.i16_typ_bandeinzug OF

				 BANDWECHSLER_V2:
					visu_hinten.in.current_visu_folie := 'BA_1700_BAND_EINFAEDELN';

				SERVO:
					visu_hinten.in.current_visu_folie := 'BA1700_SERVO_BAND_EINFAEDELN';
			END_CASE
			fb_state_entry.i16_next_step := 295;
		END_IF

(*=======================================================*)
	295:	(* Vorschub ausfahren und fertig -> Band wird jetzt im gleichen Einzug manuell eingelegt mit Einfädelprozedur in der Bestückachse *)
		IF fb_state_entry.E THEN
			zyl_bawe_vorschub.st_ctrl.in.b_ausfahren := TRUE;
		END_IF

		(*-----------------------Weiterschaltbedingungen----------------------------*)
		IF zyl_bawe_vorschub.st_ctrl.out.b_ausgefahren AND gb_ba_auto_kontroller THEN
			zyl_bawe_vorschub.st_ctrl.in.b_ausfahren := FALSE;
			st_ctrl_out.b_fertig_2 := TRUE;
			fb_state_entry.i16_next_step := BEREIT;
		END_IF

(*=======================================================*)
	300:	(* Fänger rechts ausfahren *)
		IF fb_state_entry.E THEN
			zyl_bawe_faenger_re.st_ctrl.in.b_ausfahren := TRUE;
		END_IF

		(*-----------------------Weiterschaltbedingungen----------------------------*)
		IF 	zyl_bawe_faenger_re.st_ctrl.out.b_ausgefahren AND
			gb_ba_auto_kontroller
			THEN
				zyl_bawe_faenger_re.st_ctrl.in.b_ausfahren := FALSE;
				fb_state_entry.i16_next_step := 310;
		END_IF

(*=======================================================*)
	310:	(* Halter rechts einfahren *)
		IF fb_state_entry.E THEN
			zyl_bawe_halter_re.st_ctrl.in.b_einfahren := TRUE;
		END_IF

		(*-----------------------Weiterschaltbedingungen----------------------------*)
		IF zyl_bawe_halter_re.st_ctrl.out.b_eingefahren AND gb_ba_auto_kontroller THEN
			zyl_bawe_halter_re.st_ctrl.in.b_einfahren := FALSE;
			fb_state_entry.i16_next_step := 315;
		END_IF

(*=======================================================*)
	315:	(* Spulenbremse rechts oben? *)

		(*-----------------------Weiterschaltbedingungen----------------------------*)
		IF zyl_haspel_re_abspulen.st_ctrl.out.b_ausgefahren AND gb_ba_auto_kontroller THEN
			fb_state_entry.i16_next_step := 320;
		END_IF

(*=======================================================*)
	320:	(* Querschub ausfahren -> nach links und Haspeln nach links: Haspel verschieben ausfahren und Bandabzug einfahren *)
		IF fb_state_entry.E THEN
			zyl_bawe_querschub.st_ctrl.in.b_ausfahren := TRUE;
			zyl_haspel_verschieben.st_ctrl.in.b_ausfahren := TRUE;
			zyl_bandeinzuege_verschieben.st_ctrl.in.b_einfahren := TRUE;
		END_IF

		(*-----------------------Weiterschaltbedingungen----------------------------*)
		IF 	zyl_bawe_querschub.st_ctrl.out.b_ausgefahren AND
			zyl_haspel_verschieben.st_ctrl.out.b_ausgefahren AND
			zyl_bandeinzuege_verschieben.st_ctrl.out.b_eingefahren AND
			gb_ba_auto_kontroller
			THEN
				zyl_bawe_querschub.st_ctrl.in.b_ausfahren := FALSE;
				zyl_haspel_verschieben.st_ctrl.in.b_ausfahren := FALSE;
				zyl_bandeinzuege_verschieben.st_ctrl.in.b_einfahren := FALSE;
				CASE gst_datensatz.st_wkz.i16_typ_bandeinzug OF

					BANDWECHSLER_V2:
						fb_state_entry.i16_next_step := 330;

					SERVO:
						fb_state_entry.i16_next_step := 325;
				END_CASE
		END_IF

		IF fb_state_entry.X THEN
			b_spulenwechsel := FALSE;
		END_IF

(*=======================================================*)
	325:	(* Igelrad auf Position *)
		IF fb_state_entry.E THEN
			axis_bandeinzug_achse.st_ctrl.in.b_startpos := TRUE;
			fb_ton_wz.PT := t#100ms;
			fb_ton_wz.IN := TRUE;
		END_IF

		(*-----------------------Weiterschaltbedingungen----------------------------*)
		IF axis_bandeinzug_achse.st_ctrl.out.b_servo_auf_einfaedelpos
		AND gb_ba_auto_kontroller AND fb_ton_wz.Q THEN
			axis_bandeinzug_achse.st_ctrl.in.b_startpos := FALSE;
			fb_state_entry.i16_next_step := 330;
		END_IF

		IF fb_state_entry.X THEN
			fb_ton_wz.IN := FALSE;
		END_IF

(*=======================================================*)
	330:	(* Vorschub ausfahren *)
		IF fb_state_entry.E THEN
			zyl_bawe_vorschub.st_ctrl.in.b_ausfahren := TRUE;
			i16_akt_einfaedeln := i16_akt_einfaedeln + 1;
		END_IF

		(*-----------------------Weiterschaltbedingungen----------------------------*)
		IF zyl_bawe_vorschub.st_ctrl.out.b_ausgefahren AND gb_ba_auto_kontroller THEN
			zyl_bawe_vorschub.st_ctrl.in.b_ausfahren := FALSE;
			IF i16_akt_einfaedeln < i16_vorgabe_einfaedeln THEN
				fb_state_entry.i16_next_step := 340;
			ELSE
				fb_state_entry.i16_next_step := 390;		 (*mit Wartezeit alt 400*)
			END_IF
		END_IF

(*=======================================================*)
	340:	(* Halter rechts ausfahren *)
		IF fb_state_entry.E THEN
			zyl_bawe_halter_re.st_ctrl.in.b_ausfahren := TRUE;
		END_IF

		(*-----------------------Weiterschaltbedingungen----------------------------*)
		IF zyl_bawe_halter_re.st_ctrl.out.b_ausgefahren AND gb_ba_auto_kontroller THEN
			zyl_bawe_halter_re.st_ctrl.in.b_ausfahren := FALSE;
			fb_state_entry.i16_next_step := 350;
		END_IF

(*=======================================================*)
	350:	(* Fänger rechts einfahren *)
		IF fb_state_entry.E THEN
			zyl_bawe_faenger_re.st_ctrl.in.b_einfahren := TRUE;
		END_IF

		(*-----------------------Weiterschaltbedingungen----------------------------*)
		IF zyl_bawe_faenger_re.st_ctrl.out.b_eingefahren AND gb_ba_auto_kontroller THEN
			zyl_bawe_faenger_re.st_ctrl.in.b_einfahren := FALSE;
			fb_state_entry.i16_next_step := 360;
		END_IF

(*=======================================================*)
	360:	(* Vorschub einfahren *)
		IF fb_state_entry.E THEN
			zyl_bawe_vorschub.st_ctrl.in.b_einfahren := TRUE;
		END_IF

		(*-----------------------Weiterschaltbedingungen----------------------------*)
		IF zyl_bawe_vorschub.st_ctrl.out.b_eingefahren AND gb_ba_auto_kontroller THEN
			zyl_bawe_vorschub.st_ctrl.in.b_einfahren := FALSE;
			fb_state_entry.i16_next_step := 370;
		END_IF

(*=======================================================*)
	370:	(* Fänger rechts ausfahren *)
		IF fb_state_entry.E THEN
			zyl_bawe_faenger_re.st_ctrl.in.b_ausfahren := TRUE;
		END_IF

		(*-----------------------Weiterschaltbedingungen----------------------------*)
		IF zyl_bawe_faenger_re.st_ctrl.out.b_ausgefahren AND gb_ba_auto_kontroller THEN
			zyl_bawe_faenger_re.st_ctrl.in.b_ausfahren := FALSE;
			fb_state_entry.i16_next_step := 380;
		END_IF

(*=======================================================*)
	380:	(* Halter rechts einfahren *)
		IF fb_state_entry.E THEN
			zyl_bawe_halter_re.st_ctrl.in.b_einfahren := TRUE;
		END_IF

		(*-----------------------Weiterschaltbedingungen----------------------------*)
		IF zyl_bawe_halter_re.st_ctrl.out.b_eingefahren AND gb_ba_auto_kontroller THEN
			zyl_bawe_halter_re.st_ctrl.in.b_einfahren := FALSE;
			fb_state_entry.i16_next_step := 330;
		END_IF

(*=======================================================*)
	390:	(* Wartezeit damit der Fänger vom WZ trifft*)
		IF	 fb_state_entry.E THEN
			fb_ton_wz.IN:=FALSE;
		END_IF
		fb_ton_wz(IN:=TRUE,PT:=t#1000ms);
		(*-----------------------Weiterschaltbedingungen----------------------------*)
		IF 	fb_ton_wz.Q THEN
			fb_ton_wz.IN:=FALSE;
			fb_state_entry.i16_next_step := 400;
		END_IF

(*=======================================================*)
	400:	(* Nocken für Zylinder am Bandeinzug einschalten und somit Bandfänger ausfahren bzw. Bremse an Servobandeinzug wieder fest machen. *)

		CASE gst_datensatz.st_wkz.i16_typ_bandeinzug OF

			BANDWECHSLER_V2:

				IF fb_state_entry.E THEN
					(* Bandwechsler V2 ohne Sensoren und anderen Zylindern *)
					gst_datensatz.st_wkz.nockenschaltwerk_bestueckachse.arr_nocken[NO_BW_BANDFAENGER_BAWEV2_EINFAHREN].b_camvalid := TRUE;
					gst_datensatz.st_wkz.nockenschaltwerk_bestueckachse.arr_nocken[NO_BW_BANDFAENGER_BAWEV2_AUSFAHREN].b_camvalid := TRUE;
					gst_datensatz.st_wkz.nockenschaltwerk_bestueckachse.arr_nocken[NO_BW_BANDKLEMMEN_BAWEV2_EINFAHREN].b_camvalid := TRUE;
					gst_datensatz.st_wkz.nockenschaltwerk_bestueckachse.arr_nocken[NO_BW_BANDKLEMMEN_BAWEV2_AUSFAHREN].b_camvalid := TRUE;

					gst_datensatz.st_wkz.nockenschaltwerk_bestueckachse.arr_nocken[NO_PNEUMATIKBANDEINZUG_GLS].b_camvalid := TRUE;

					zyl_bandfaenger.fb.b_no_gesteuert_im_norm_betrieb := FALSE;
					zyl_bandklemmen.fb.b_no_gesteuert_im_norm_betrieb := FALSE;
					fb_ton_wz.PT := t#500ms;
					fb_ton_wz.IN := TRUE;
				END_IF

				(*-----------------------Weiterschaltbedingungen----------------------------*)
				IF fb_ton_wz.Q THEN
					fb_ton_wz.IN := FALSE;
					fb_state_entry.i16_next_step := 410;
				END_IF

			SERVO:
				IF fb_state_entry.E THEN
					axis_bandeinzug_achse.st_ctrl.in.b_bremse_auf := TRUE;	(* Bremse auf zum Position übernehmen *)
				END_IF

				(*-----------------------Weiterschaltbedingungen----------------------------*)
				IF axis_bandeinzug_achse.st_ctrl.out.b_bremse_geoeffnet THEN
					axis_bandeinzug_achse.st_ctrl.in.b_bremse_auf := FALSE;
					fb_state_entry.i16_next_step := 410;
				END_IF
		END_CASE;

(*=======================================================*)
	410:	(* Fänger rechts einfahren *)
		IF fb_state_entry.E THEN
			zyl_bawe_faenger_re.st_ctrl.in.b_einfahren := TRUE;
		END_IF

		(*-----------------------Weiterschaltbedingungen----------------------------*)
		IF zyl_bawe_faenger_re.st_ctrl.out.b_eingefahren
		AND gb_ba_auto_kontroller THEN
			zyl_bawe_faenger_re.st_ctrl.in.b_einfahren := FALSE;
			(* Bandwechsel ist fertig *)
			st_ctrl_out.b_fertig := TRUE;
			fb_state_entry.i16_next_step := BEREIT;
		END_IF


(*---------------------------------------------------------------------------------------------------------------------------------------------------------------------------------------------------*)
(*========================Bandeinzug rechts ist leer===============================*)
	500:	(* Fänger links ausfahren zum Band halten, Fänger rechts einfahren zur Bandfreigabe im rechten Einzug - Halter gegensinnig *)
		IF fb_state_entry.E THEN
			zyl_bawe_faenger_re.st_ctrl.in.b_ausfahren := TRUE;
			zyl_bawe_faenger_li.st_ctrl.in.b_einfahren := TRUE;
			zyl_bawe_halter_re.st_ctrl.in.b_einfahren := TRUE;
			zyl_bawe_halter_li.st_ctrl.in.b_ausfahren := TRUE;
		END_IF

		(*-----------------------Weiterschaltbedingungen----------------------------*)
		IF 	zyl_bawe_faenger_re.st_ctrl.out.b_ausgefahren AND
			zyl_bawe_faenger_li.st_ctrl.out.b_eingefahren AND
			zyl_bawe_halter_re.st_ctrl.out.b_eingefahren AND
			zyl_bawe_halter_li.st_ctrl.out.b_ausgefahren AND
			gb_ba_auto_kontroller
			THEN
				zyl_bawe_faenger_re.st_ctrl.in.b_ausfahren := FALSE;
				zyl_bawe_faenger_li.st_ctrl.in.b_einfahren := FALSE;
				zyl_bawe_halter_re.st_ctrl.in.b_einfahren := FALSE;
				zyl_bawe_halter_li.st_ctrl.in.b_ausfahren := FALSE;
				fb_state_entry.i16_next_step := 510;
		END_IF

(*=======================================================*)
	510:	(* Band-Zylinder einfahren bzw. Servobandeinzug lösen *)
		CASE gst_datensatz.st_wkz.i16_typ_bandeinzug OF
			BANDWECHSLER_V2:
				IF fb_state_entry.E THEN
					(* Zylinder einfahren *)
					zyl_bandfaenger.st_ctrl.in.b_einfahren := TRUE;
					zyl_bandklemmen.st_ctrl.in.b_einfahren := TRUE;
				END_IF

				(*-----------------------Weiterschaltbedingungen----------------------------*)
				IF 	zyl_bandfaenger.st_ctrl.out.b_eingefahren AND
					zyl_bandklemmen.st_ctrl.out.b_eingefahren AND
					gb_ba_auto_kontroller
					THEN
						zyl_bandfaenger.st_ctrl.in.b_einfahren := FALSE;
						zyl_bandklemmen.st_ctrl.in.b_einfahren := FALSE;
						fb_state_entry.i16_next_step := 520;
				END_IF

			SERVO:
				zyl_bawe_faenger_re.st_ctrl.in.b_einfahren := TRUE;
				zyl_bawe_halter_re.st_ctrl.in.b_einfahren := TRUE;
				(*-----------------------Weiterschaltbedingungen----------------------------*)
				IF 	zyl_bawe_faenger_re.st_ctrl.out.b_eingefahren AND
					zyl_bawe_halter_re.st_ctrl.out.b_eingefahren AND
					gb_ba_auto_kontroller
					THEN
						zyl_bawe_faenger_re.st_ctrl.in.b_einfahren := FALSE;
						zyl_bawe_halter_re.st_ctrl.in.b_einfahren := FALSE;
						fb_state_entry.i16_next_step := 516;
				END_IF
		END_CASE;

(*=======================================================*)
	516:	(* Servobandeinzug rückwärts fahren, damit die Ausschiebezylinder das Band sicher erwischen *)
		IF fb_state_entry.E THEN
			axis_bandeinzug_achse.st_ctrl.in.b_ausfaedeln_servo := TRUE;
		END_IF

		(*-----------------------Weiterschaltbedingungen----------------------------*)
		IF axis_bandeinzug_achse.st_ctrl.out.b_ausgefaedelt_servo AND NOT fb_state_entry.E THEN
			axis_bandeinzug_achse.st_ctrl.in.b_ausfaedeln_servo := FALSE;
			fb_state_entry.i16_next_step := 517;(*Neu*)
		END_IF

(*=======================================================*)
	517:	(* Fänger ins Band fahren, damit die Bremse gelöst werden kann *)
		IF fb_state_entry.E THEN
				zyl_bawe_faenger_re.st_ctrl.in.b_ausfahren := TRUE;
		END_IF

		(*-----------------------Weiterschaltbedingungen----------------------------*)
		IF 	zyl_bawe_faenger_re.st_ctrl.out.b_ausgefahren AND
			gb_ba_auto_kontroller
			THEN
				zyl_bawe_faenger_re.st_ctrl.in.b_ausfahren := FALSE;
				fb_state_entry.i16_next_step := 518;
		END_IF

(*=======================================================*)
	518:	(* Bremse an Servobandeinzug lösen, damit Band heraus gezogen werden kann. Die Bestückachse hat die Slavekopplung bereits gelöst. *)
		IF fb_state_entry.E THEN
			axis_bandeinzug_achse.st_ctrl.in.b_bremse_auf := TRUE;
		END_IF

		(*-----------------------Weiterschaltbedingungen----------------------------*)
		IF axis_bandeinzug_achse.st_ctrl.out.b_bremse_geoeffnet AND NOT fb_state_entry.E THEN
			axis_bandeinzug_achse.st_ctrl.in.b_bremse_auf := FALSE;
			fb_state_entry.i16_next_step := 520;
		END_IF

(*=======================================================*)
	520:	(* Vorschub einfahren und Band aus WKZ rausziehen *)
		IF fb_state_entry.E THEN
			zyl_bawe_vorschub.st_ctrl.in.b_einfahren := TRUE;
			i16_akt_ausfaedeln := i16_akt_ausfaedeln + 1;
		END_IF

		(*-----------------------Weiterschaltbedingungen----------------------------*)
		IF zyl_bawe_vorschub.st_ctrl.out.b_eingefahren AND gb_ba_auto_kontroller THEN
			zyl_bawe_vorschub.st_ctrl.in.b_einfahren := FALSE;
			IF i16_akt_ausfaedeln <= i16_vorgabe_ausfaedeln THEN
				fb_state_entry.i16_next_step := 530;
			ELSE
				fb_state_entry.i16_next_step := 580;
			END_IF
		END_IF

(*=======================================================*)
	530:	(* Bandwechselhalter rechts ausfahren um Band nachfassen zu können *)
		IF fb_state_entry.E THEN
			zyl_bawe_halter_re.st_ctrl.in.b_ausfahren := TRUE;
		END_IF

		(*-----------------------Weiterschaltbedingungen----------------------------*)
		IF zyl_bawe_halter_re.st_ctrl.out.b_ausgefahren AND gb_ba_auto_kontroller THEN
			zyl_bawe_halter_re.st_ctrl.in.b_ausfahren := FALSE;
			fb_state_entry.i16_next_step := 540;
		END_IF

(*=======================================================*)
	540:	(* Bandwechselfänger rechts einfahren*)
		IF fb_state_entry.E THEN
			zyl_bawe_faenger_re.st_ctrl.in.b_einfahren := TRUE;
		END_IF

		(*-----------------------Weiterschaltbedingungen----------------------------*)
		IF zyl_bawe_faenger_re.st_ctrl.out.b_eingefahren AND gb_ba_auto_kontroller THEN
			zyl_bawe_faenger_re.st_ctrl.in.b_einfahren := FALSE;
			fb_state_entry.i16_next_step := 550;
		END_IF

(*=======================================================*)
	550:	(* Vorschub ausfahren und Band nachfassen *)
		IF fb_state_entry.E THEN
			zyl_bawe_vorschub.st_ctrl.in.b_ausfahren := TRUE;
		END_IF

		(*-----------------------Weiterschaltbedingungen----------------------------*)
		IF zyl_bawe_vorschub.st_ctrl.out.b_ausgefahren AND gb_ba_auto_kontroller THEN
			zyl_bawe_vorschub.st_ctrl.in.b_ausfahren := FALSE;
			fb_state_entry.i16_next_step := 560;
		END_IF

(*=======================================================*)
	560:	(* Bandwechselfänger rechts ausfahren zum Band halten *)
		IF fb_state_entry.E THEN
			zyl_bawe_faenger_re.st_ctrl.in.b_ausfahren := TRUE;
		END_IF

		(*-----------------------Weiterschaltbedingungen----------------------------*)
		IF zyl_bawe_faenger_re.st_ctrl.out.b_ausgefahren AND gb_ba_auto_kontroller THEN
			zyl_bawe_faenger_re.st_ctrl.in.b_ausfahren := FALSE;
			fb_state_entry.i16_next_step := 570;
		END_IF

(*=======================================================*)
	570:	(* Bandwechselhalter rechts einfahren und Band freigeben*)
		IF fb_state_entry.E THEN
			zyl_bawe_halter_re.st_ctrl.in.b_einfahren := TRUE;
		END_IF

		(*-----------------------Weiterschaltbedingungen----------------------------*)
		IF zyl_bawe_halter_re.st_ctrl.out.b_eingefahren AND gb_ba_auto_kontroller THEN
			zyl_bawe_halter_re.st_ctrl.in.b_einfahren := FALSE;
			fb_state_entry.i16_next_step := 520;
		END_IF

(*=======================================================*)
	580:	(* Fänger rechts einfahren zum Ausfädeln *)
		IF fb_state_entry.E THEN
			zyl_bawe_faenger_re.st_ctrl.in.b_einfahren := TRUE;
		END_IF

		(*-----------------------Weiterschaltbedingungen----------------------------*)
		IF 	zyl_bawe_faenger_re.st_ctrl.out.b_eingefahren AND
			gb_ba_auto_kontroller
			THEN
				zyl_bawe_faenger_re.st_ctrl.in.b_einfahren := FALSE;
				fb_state_entry.i16_next_step := 590;
		END_IF

(*=======================================================*)
	590:	(* Band ist herausgezogen  - prüfe Einstellung bzw. Bandanwesenheit im linken Einzug *)
		b_ausgefaedelt:=b_materialmangel;
		(*-----------------------Weiterschaltbedingungen----------------------------*)
		IF fb_tof_bandende_li.Q  AND gst_datensatz.st_md.b_auto_Bandwechsel THEN
			b_spulenwechsel := TRUE;
			fb_state_entry.i16_next_step := 600;
		ELSE
			(* Bandherausziehen ist fertig *)
			fb_state_entry.i16_next_step := 595;
		END_IF

(*=======================================================*)
	591:	(* Bediener muss am Backpanel auswählen ob Bandwechsel oder Trennstelle *)

		(*-----------------------Weiterschaltbedingungen----------------------------*)
		IF visu_hinten.out.b_Bandwechsel THEN
			(* Band vorhanden -> Beginn automatischer Bandwechsel *)
			visu_hinten.in.b_bandwechsel_aktiv := FALSE;
			visu_hinten.in.current_visu_folie := 'BESTUECKZELLE_1700';
			fb_state_entry.i16_next_step := 600;
		ELSIF visu_hinten.out.b_Trennstelle THEN
			visu_hinten.in.b_bandwechsel_aktiv := FALSE;
			CASE gst_datensatz.st_wkz.i16_typ_bandeinzug OF

				BANDWECHSLER_V2:
					visu_hinten.in.current_visu_folie := 'BA_1700_BAND_EINFAEDELN';

				SERVO:
					visu_hinten.in.current_visu_folie := 'BA1700_SERVO_BAND_EINFAEDELN';
			END_CASE
			fb_state_entry.i16_next_step := 595;
		END_IF


(*=======================================================*)
	595:	(* Vorschub ausfahren und fertig -> Band wird jetzt im gleichen Einzug manuell eingelegt mit Einfädelprozedur in der Bestückachse *)
		IF fb_state_entry.E THEN
			zyl_bawe_vorschub.st_ctrl.in.b_ausfahren := TRUE;
		END_IF

		(*-----------------------Weiterschaltbedingungen----------------------------*)
		IF zyl_bawe_vorschub.st_ctrl.out.b_ausgefahren AND gb_ba_auto_kontroller THEN
			zyl_bawe_vorschub.st_ctrl.in.b_ausfahren := FALSE;
			st_ctrl_out.b_fertig_2 := TRUE;
			fb_state_entry.i16_next_step := BEREIT;
		END_IF

(*=======================================================*)
	600:	(* Fänger links ausfahren *)
		IF fb_state_entry.E THEN
			zyl_bawe_faenger_li.st_ctrl.in.b_ausfahren := TRUE;
		END_IF

		(*-----------------------Weiterschaltbedingungen----------------------------*)
		IF 	zyl_bawe_faenger_li.st_ctrl.out.b_ausgefahren AND
			gb_ba_auto_kontroller
			THEN
				zyl_bawe_faenger_li.st_ctrl.in.b_ausfahren := FALSE;
				fb_state_entry.i16_next_step := 610;
		END_IF

(*=======================================================*)
	610:	(* Halter links einfahren *)
		IF fb_state_entry.E THEN
			zyl_bawe_halter_li.st_ctrl.in.b_einfahren := TRUE;
		END_IF

		(*-----------------------Weiterschaltbedingungen----------------------------*)
		IF zyl_bawe_halter_li.st_ctrl.out.b_eingefahren AND gb_ba_auto_kontroller THEN
			zyl_bawe_halter_li.st_ctrl.in.b_einfahren := FALSE;
			fb_state_entry.i16_next_step := 615;
		END_IF

(*=======================================================*)
	615:	(* Spulenbremse links oben? *)

		(*-----------------------Weiterschaltbedingungen----------------------------*)
		IF zyl_haspel_li_abspulen.st_ctrl.out.b_ausgefahren AND gb_ba_auto_kontroller THEN
			fb_state_entry.i16_next_step := 620;
		END_IF

(*=======================================================*)
	620:	(* Querschub einfahren -> nach rechts und Haspeln nach rechts: Haspel verschieben einfahren und Bandabzug ausfahren*)
		IF fb_state_entry.E THEN
			zyl_bawe_querschub.st_ctrl.in.b_einfahren := TRUE;
			zyl_haspel_verschieben.st_ctrl.in.b_einfahren := TRUE;
			zyl_bandeinzuege_verschieben.st_ctrl.in.b_ausfahren := TRUE;
		END_IF

		(*-----------------------Weiterschaltbedingungen----------------------------*)
		IF 	zyl_bawe_querschub.st_ctrl.out.b_eingefahren AND
			zyl_haspel_verschieben.st_ctrl.out.b_eingefahren AND
			zyl_bandeinzuege_verschieben.st_ctrl.out.b_ausgefahren AND
			gb_ba_auto_kontroller
			THEN
				zyl_bawe_querschub.st_ctrl.in.b_einfahren := FALSE;
				zyl_haspel_verschieben.st_ctrl.in.b_einfahren := FALSE;
				zyl_bandeinzuege_verschieben.st_ctrl.in.b_ausfahren := FALSE;
				CASE gst_datensatz.st_wkz.i16_typ_bandeinzug OF

					BANDWECHSLER_V2:
						fb_state_entry.i16_next_step := 630;

					SERVO:
						fb_state_entry.i16_next_step := 625;
				END_CASE
		END_IF

		IF fb_state_entry.X THEN
			b_spulenwechsel := FALSE;
		END_IF

(*=======================================================*)
	625:	(* Igelrad auf Position *)
		IF fb_state_entry.E THEN
			axis_bandeinzug_achse.st_ctrl.in.b_startpos := TRUE;
			fb_ton_wz.PT := t#100ms;
			fb_ton_wz.IN := TRUE;
		END_IF

		(*-----------------------Weiterschaltbedingungen----------------------------*)
		IF axis_bandeinzug_achse.st_ctrl.out.b_servo_auf_einfaedelpos
			AND gb_ba_auto_kontroller AND fb_ton_wz.Q THEN
			axis_bandeinzug_achse.st_ctrl.in.b_startpos := FALSE;
			fb_state_entry.i16_next_step := 630;
		END_IF

		IF fb_state_entry.X THEN
			fb_ton_wz.IN := FALSE;
		END_IF

(*=======================================================*)
	630:	(* Vorschub ausfahren *)
		IF fb_state_entry.E THEN
			zyl_bawe_vorschub.st_ctrl.in.b_ausfahren := TRUE;
			i16_akt_einfaedeln := i16_akt_einfaedeln + 1;
		END_IF

